(* CODESYS project CodesysJsonParser

Project tree, tasks and I/O mapping:
  Device : ctrlX CORE x64, Bosch Rexroth AG, version 3.6.3.0
    application Application
      libraries: ; ADT, 1.0.0 (Open Source); FloatingPointUtils, 3.5.17.0 (System)
      task MainTask (cyclic, interval 10 ms, priority 30) calls PLC_PRG
      CheckFunctions/
        function CheckBounds [ST]
        function CheckDivDInt [ST]
        function CheckDivLInt [ST]
        function CheckDivLReal [ST]
        function CheckDivReal [ST]
        function CheckLRangeSigned [ST]
        function CheckLRangeUnsigned [ST]
        function CheckPointer [ST]
        function CheckRangeSigned [ST]
        function CheckRangeUnsigned [ST]
      DynamicInterfaces (Not Yet Tested)/
        interface iDynamicDataContainer
        interface iDynamicHashTable
      function GetJsonNodeByKey2 [ST]
      function GetJsonNodeByKey [ST]
      function GetNextJsonToken [ST]
      function GetNodeAsBool [ST]
      function GetNodeAsInt [ST]
      function GetNodeAsObject [ST]
      function GetNodeAsReal [ST]
      function GetNodeAsString [ST]
      function GetNodeAtIndex [ST]
      function GetSubString [ST]
      data type HashData
      function isJsonNodeNull [ST]
      Json/
        function block FB_JsonDomParser [ST]: CopyJson, CopyString, FindMember, GetArrayValueByIdx, GetBool, GetInt, GetString, ParseDocument
        function block FB_JsonSaxWriter [ST]: AddBool, AddDint, AddKey, AddNull, AddString, AddUdint, CopyDocument, EndArray, EndObject, FB_Exit, Init, ResetDocument, StartArray, StartObject
        Types/
      data type JsonDataType
      function block JsonDomParser [ST]: CopyJson, CopyString, FB_Exit, FindMember, GetArrayValueByIdx, GetBool, GetInt, GetReal, GetString, isNull, ParseDocument, ResetDocument
      function JsonHadlr [ST]
      data type JsonObject
      function block JsonParser2 [ST]: CreateJsonType, DeleteJsonNode, FB_Exit, GetRootDoc, Parse, Clean, CreateArray, CreateObj
      function block JsonParser [ST]: Clean, DeleteJsonNode, FB_Exit, GetRootDoc, Parse
      function block JsonSaxWriter [ST]: AddBool, AddChild, AddDint, AddFloat, AddKey, AddNull, AddString, AddUdint, Clean, CopyDocument, CreateArray, CreateJsonType, CreateObj, DeleteJsonNode, EndArray, EndObject, GetRoot, Init, ResetDocument, StartArray, StartObject
      data type JsonSerializeConfig
      data type JsonToken
      data type JsonTokenType
      data type JsonType
      global variables Parameters
      data type pDoc
      program PLC_PRG [ST]
      data type pVoid
      ResizableMem (Not Fully Tested)/
        function block DynamicHashContainer [ST]: CopyToNew, EndResize, FB_Exit, Get, GetNew, GetNewPointer, GetPointer, GetSize, Put, StartResize, FB_Init
        function block DynamicHashTable [ST]: EndResize
        function block DynamicMap [ST]: Remove, Get, HasKey, Put, Resize, Size
        function block DynamicQueue [ST]
        function block DynamicStringContainer [ST]: FB_Exit, CopyToNew, EndResize, Get, GetNew, GetNewPointer, GetPointer, Put
        function block JsonListManager [ST]: Create, Destroy, GetAt, Push
        function block DynamicJsonContainerContainer [ST]: CopyToNew, EndResize, FB_Exit, Get, GetNew, GetNewPointer, GetPointer, GetSize, Put, FB_Init, StartResize
        function block DynamicJsonObjectContainer [ST]: CopyToNew, FB_Exit, Get, GetNew, GetNewPointer, GetPointer, Put, EndResize, FB_Init, GetSize, StartResize
        function block DynamicJsonTypeContainer [ST]: CopyToNew, EndResize, FB_Init, Get, GetNew, GetNewPointer, GetPointer, Put, FB_Exit, GetSize, StartResize
        function block DynamicList [ST]: Get, GetPointer, Insert, Pop, PopBack, PopFront, PushBack, PushFront, Put, Remove, Resize
        global variables JsonHelpers
        function block JsonObjectManager [ST]: Create, Destroy, GetKeyAtIndex, GetValue, Put, Size, FB_Exit
      Serialize/
        function JsonSerializer [ST]
        function SerializeJsonValue [ST]
        function WriteDint [ST]
        function WriteNewLine [ST]
        function WriteReal [ST]
        global variables SerializerConstants
        function WriteByte [ST]
        function WriteColon [ST]
        function WriteEscapedString [ST]
        function WriteIndent [ST]
      Symbols
      Util/
        function block ADT_CompareString [ST]: Compare
        function block StringHash [ST]: Hash
    Realtime_Data : DataLayer, Bosch Rexroth AG, version 3.6.2.0
  commdata.all
  JsonST.Sync
*)

// Device/Application/HashData
{attribute 'enable_dynamic_creation'}
(*Data to keep track of Hash Table to ensure collisions are handled gracefully*)
TYPE HashData :
STRUCT
	isOccupied : BOOL; 
	isDeleted  : BOOL; 
END_STRUCT
END_TYPE

// Device/Application/JsonDataType
TYPE JsonDataType :
(
    JSON_DATA_NULL,
    JSON_DATA_BOOL,
    JSON_DATA_INT,
    JSON_DATA_REAL,
    JSON_DATA_STRING,
    JSON_DATA_ARRAY,
    JSON_DATA_OBJECT
);
END_TYPE

// Device/Application/JsonObject
{attribute 'enable_dynamic_creation'}
TYPE JsonObject :
STRUCT
	pKeys   : POINTER TO POINTER TO JsonType; 
	pValues : POINTER TO  POINTER TO JsonType; 
	iNumValues : INT; 
END_STRUCT
END_TYPE

// Device/Application/JsonSerializeConfig
TYPE JsonSerializeConfig :
STRUCT
    PrettyPrint  : BOOL;        // Enable pretty printing
    IndentLevel  : DINT;        // Current indentation depth (pass 0 initially)
    IndentSize   : DINT;        // Number of spaces per indent level
END_STRUCT
END_TYPE

// Device/Application/JsonToken
TYPE JsonToken :
STRUCT
	TokenType : JsonTokenType;
    StartIndex : LINT;
    Length : DINT;
END_STRUCT
END_TYPE

// Device/Application/JsonTokenType
TYPE JsonTokenType :
(
	JSON_TOKEN_NULL,
    JSON_TOKEN_TRUE,
    JSON_TOKEN_FALSE,
    JSON_TOKEN_NUMBER,
    JSON_TOKEN_STRING,
    JSON_TOKEN_LBRACE,      // {
    JSON_TOKEN_RBRACE,      // }
    JSON_TOKEN_LBRACKET,    // [
    JSON_TOKEN_RBRACKET,    // ]
    JSON_TOKEN_COMMA,       // ,
    JSON_TOKEN_COLON,       // :
    JSON_TOKEN_EOF,
    JSON_TOKEN_ERROR
);
END_TYPE

// Device/Application/JsonType
{attribute 'enable_dynamic_creation'}
TYPE JsonType :
STRUCT
	DataType : JsonDataType; 
	pValue   : pVoid; 
END_STRUCT
END_TYPE

// Device/Application/pDoc
TYPE pDoc : __XWORD; END_TYPE

// Device/Application/pVoid
{attribute 'enable_dynamic_creation'}
TYPE pVoid : __XWORD; END_TYPE

// Device/Application/Parameters
{attribute 'qualified_only'}
VAR_GLOBAL CONSTANT
	MAX_DOC_DEPTH : INT := 50; 
	MAX_ARR_SIZE : INT := 50; 
END_VAR

// Device/Application/ResizableMem (Not Fully Tested)/JsonHelpers
{attribute 'qualified_only'}
VAR_GLOBAL
	instStrCompare     : ADT_CompareString; 
	instStrHash        : StringHash; 
END_VAR

// Device/Application/Serialize/SerializerConstants
{attribute 'qualified_only'}
VAR_GLOBAL CONSTANT
	INDENT_CHAR : BYTE := 32;   // space
    INDENT_SIZE : DINT := 4;    // 4 spaces per level
    NEWLINE_CR  : BYTE := 13;   // \r
    NEWLINE_LF  : BYTE := 10;   // \n
    QUOTE       : BYTE := 34;   // "
    BACKSLASH   : BYTE := 92;   // \
    COLON       : BYTE := 58;   // :
    COMMA       : BYTE := 44;   // ,
    NULL_TERM   : BYTE := 0;    // null terminator
	START_OBJ    : BYTE := 123; 
	END_OBJ      : BYTE := 125; 
	START_ARR    : BYTE := 91; 
	END_ARR      : BYTE := 93;
END_VAR

// Device/Application/PLC_PRG
PROGRAM PLC_PRG
VAR
	Parser : JsonParser2; 
	jsonInput: STRING(8192) := '{"name":"Test","value":42,"active":true, "RealValue" : 12.8, "arrTest" : [[10,11,15][10,11,12]], "subObject" : {"subVal" : 10}}';
	pJson: POINTER TO JsonType;
	pDoc : POINTER TO JsonObject; 
	bVal: BOOL;
	strVal : STRING; 
	size: UDINT;
	iValue: LINT;
	rValue: REAL;
	pJsonAr: POINTER TO JsonType;
	val2: DINT;
	pDoc2 : POINTER TO JsonObject; 
	iVal3: DINT;
	pJsonObject: POINTER TO JsonObjectManager;
	pDint: POINTER TO DINT;
	pByte: Pointer TO Byte;
	pDint2: POINTER TO DINT;
	JsonSettings : JsonSerializeConfig; 
	jSonString : STRING(1000);
	jSonString2 : STRING(1000); 
	Writer : JsonSaxWriter; 
END_VAR

Parser.Parse(ADR(jsonInput),SIZEOF(jsonInput));
pDoc := Parser.GetRootDoc(); 
pJson := GetJsonNodeByKey2('active', pDoc := pDoc); 
GetNodeAsBool(pJson, bJsonVal => bVal); 
pJson := GetJsonNodeByKey2('name',pDoc := pDoc); 
GetNodeAsString(pJson, ADR(strVal),SIZEOF(strVal),retStrSize => size); 
pJson := GetJsonNodeByKey2('value',pDoc); 
GetNodeAsInt(pJson, iJsonVal => iValue); 
pJson := GetJsonNodeByKey2('RealValue',pDoc);
GetNodeAsReal(pJson, rJsonVal => rValue); 
pJson := GetJsonNodeByKey2('arrTest',pDoc); 
pJsonAr := GetNodeAtIndex(pJson,1); 
pJsonAr := GetNodeAtIndex(pJsonAr,2); 
GetNodeAsInt(pJsonAr, iJsonVal => val2); 
pDOC2 := GetJsonNodeByKey2('subObject', pDoc := pDoc);  
pJson := GetJsonNodeByKey2('subVal', pDoc := pDoc2); 
GetNodeAsInt(pJson, iJsonVal => iVal3); 

JsonSettings.IndentSize := 4; 
JsonSettings.PrettyPrint := TRUE; 
JsonSerializer(pDOc, ADR(jSonString),SIZEOF(JsonString),JsonSettings); 
Parser.Clean();
Writer.StartObject(); 
Writer.AddKey('test_bool'); 
Writer.AddBool(TRUE); 
Writer.AddKey('test_dint'); 
Writer.AddDint(100); 
Writer.AddKey('test_real'); 
Writer.AddFloat(90.2); 
Writer.AddKey('test_null'); 
Writer.AddNull(); 
Writer.AddKey('test_string'); 
Writer.AddString('test string val'); 
Writer.AddKey('test_arr'); 
Writer.StartArray(); 
	Writer.StartArray();
		Writer.AddDint(1); 
		Writer.AddDint(2); 
		Writer.AddDint(3);
	Writer.EndArray(); 
	Writer.StartArray(); 
		Writer.AddDint(4); 
		Writer.AddDint(5); 
		Writer.AddDint(6); 
	Writer.EndArray();  
Writer.EndArray(); 
Writer.AddKey('test_obj'); 
Writer.StartObject(); 
	Writer.AddKey('test_internal_object');
	Writer.StartObject(); 
		Writer.AddKey('test_obj_val'); 
		Writer.AddString('obj_val'); 
		Writer.AddKey('test2'); 
		Writer.AddDint(1); 
	Writer.EndObject(); 
	Writer.AddKey('test_internal_object2');
	Writer.StartObject(); 
		Writer.AddKey('test_obj_val'); 
		Writer.AddString('obj_val2'); 
		Writer.AddKey('test2'); 
		Writer.AddDint(2); 
	Writer.EndObject(); 
Writer.EndObject(); 
Writer.CopyDocument(pDoc := JsonString2, nDoc := SIZEOF(JsonString2),bPretty := TRUE); 
Writer.ResetDocument();

END_PROGRAM

// Device/Application/GetJsonNodeByKey2
FUNCTION GetJsonNodeByKey2: Pointer TO JsonType; 
VAR_INPUT
	strKey : STRING; 
END_VAR
VAR_IN_OUT
	pDoc : POINTER TO JsonType; 
END_VAR
VAR_OUTPUT
END_VAR
VAR
	i: INT;
	pStr : POINTER TO STRING; 
	pJsonObject : Pointer TO JsonObjectManager; 
END_VAR

GetJsonNodeByKey2 := 0; 
IF pDoc = 0 THEN 
	RETURN; 
END_IF
IF pDoc^.DataType <> JsonDataType.JSON_DATA_OBJECT THEN 
	RETURN; 
END_IF
pJsonObject := pDoc^.pValue; 
IF pJsonObject <> 0 THEN 
	GetJsonNodeByKey2 := pJsonObject^.GetValue(strKey); 
END_IF

END_FUNCTION

// Device/Application/ResizableMem (Not Fully Tested)/JsonObjectManager
{attribute 'enable_dynamic_creation'}
FUNCTION_BLOCK JsonObjectManager
VAR_INPUT
END_VAR
VAR
	_KeyBacking: POINTER TO DynamicStringContainer;
	_HashBacking: POINTER TO DynamicHashContainer;
	_ValueContainer: POINTER TO DynamicJsonTypeContainer;
	_HashTable: POINTER TO DynamicHashTable;
	_DynamicMap: POINTER TO DynamicMap;
	_KeysListBacking : POINTER TO DynamicStringContainer; 
	_lKeys           : POINTER TO DynamicList;
END_VAR

METHOD Create : BOOL
VAR_INPUT
END_VAR
IF _KeyBacking <> 0 THEN 
	RETURN; 
END_IF
_KeyBacking := __NEW(DynamicStringContainer(udSize := 3)); 
_HashBacking := __NEW(DynamicHashContainer(udSize :=3)); 
_ValueContainer := __NEW(DynamicJsonTypeContainer(udSize :=3)); 
_HashTable := __NEW(DynamicHashTable()); 
_HashTable^(KeyContainer := _KeyBacking^, HashDataContainer := _HashBacking^, Compareator := JsonHelpers.instStrCompare, Hasher := JsonHelpers.instStrHash); 
_DynamicMap := __NEW(DynamicMap); 
_DynamicMap^(KeyContainer := _HashTable^, ValueContainer := _ValueContainer^); 

_KeysListBacking := __NEW(DynamicStringContainer(udSize := 3));  
_lKeys           := __NEW(DynamicList); 
_lKeys^(DataContainer :=_KeysListBacking^);
END_METHOD

METHOD Destroy : BOOL
VAR_INPUT
END_VAR
IF (_KeyBacking <> 0 ) THEN 
	__DELETE(_KeyBacking);
END_IF
IF _HashBacking <> 0 THEN 
__DELETE(_HashBacking); 
END_IF
IF _ValueContainer <> 0 THEN 
__DELETE(_ValueContainer);
END_IF
IF _HashTable <> 0 THEN   
__DELETE(_HashTable); 
END_IF
IF _DynamicMap <> 0 THEN 
__DELETE(_DynamicMap); 
END_IF
IF _lKeys <> 0 THEN 
	__DELETE(_lKeys); 
END_IF
IF _KeysListBacking <> 0 THEN
	__DELETE(_KeysListBacking);
END_IF
END_METHOD

METHOD GetKeyAtIndex : Pointer TO STRING
VAR_INPUT
	index : UDINT; 
END_VAR
VAR
	pString : POINTER TO STRING; 
END_VAR
_lKeys^.Get(index,ADR(pString)); 
GetKeyAtIndex := pString;
END_METHOD

METHOD GetValue : POINTER TO JsonType
VAR_INPUT
	stKey  : STRING; 
END_VAR
VAR
	pJsonValue : POINTER TO JsonType;  
	pString : POINTER TO STRING; 
	ppString : POINTER TO POINTER TO STRING; 
END_VAR
GetValue := 0; 
pString := ADR(stKey); 
ppSTring := ADR(pString); 
IF _DynamicMap <> 0 THEN
	_DynamicMap^.Get(ppstring, ADR(pJsonValue)); 
	GetValue := pJsonValue; 
END_IF
END_METHOD

METHOD Put : BOOL
VAR_INPUT
	pString : POINTER TO BYTE; 
	pValue  : Pointer TO JsonType; 
END_VAR
Put := FALSE; 
IF _DynamicMap = 0 THEN 
	RETURN;
END_IF
IF(_DynamicMap^.Put(pKey := ADR(pString), pValue := ADR(pValue))) THEN
	_lKeys^.PushBack(ADR(pString));
	Put := TRUE;  
END_IF
END_METHOD

PROPERTY Size : UDINT
GET
IF _lKeys <> 0 THEN
	Size := _lKeys^.Size;
ELSE
	Size := 0; 
END_IF;
END_GET
END_PROPERTY

//FB_Exit must be implemented explicitly. If there is an implementation, then the
//method is called before the controller removes the code of the function block instance
//(implicit call). The return value is not evaluated.
METHOD FB_Exit: BOOL
VAR_INPUT
    bInCopyCode: BOOL;  // TRUE: the exit method is called in order to leave the instance which will be copied afterwards (online change).  
END_VAR
Destroy();
END_METHOD

END_FUNCTION_BLOCK

// Device/Application/ResizableMem (Not Fully Tested)/DynamicStringContainer
{attribute 'enable_dynamic_creation'}
FUNCTION_BLOCK DynamicStringContainer IMPLEMENTS iDynamicDataContainer
VAR_INPUT
	udSize : UDINT; 
END_VAR
VAR_OUTPUT
END_VAR
VAR
	_ptrBackingArray : POINTER TO POINTER TO BYTE;
	_ptrTempNewArray : POINTER TO POINTER TO BYTE;  
	_size : UDINT; 
	_tData : POINTER TO BYTE; 
	_pData : POINTER TO POINTER TO BYTE; 
	_newSize: UDINT;
	_byteSize : UDINT; 
END_VAR

_byteSize := SIZEOF(_tData); 
_newSize := udSize * _byteSize;
_ptrBackingArray := __NEW(BYTE,_newSize); 
_size := udSize;

//FB_Exit must be implemented explicitly. If there is an implementation, then the
//method is called before the controller removes the code of the function block instance
//(implicit call). The return value is not evaluated.
METHOD FB_Exit: BOOL
VAR_INPUT
    bInCopyCode: BOOL;  // TRUE: the exit method is called in order to leave the instance which will be copied afterwards (online change).  
END_VAR
VAR
	i: UDINT;
END_VAR
IF _ptrBackingArray <> 0 THEN 
	__DELETE(_ptrBackingArray); 
END_IF
IF _ptrTempNewArray <> 0 THEN 
	__DELETE(_ptrTempNewArray); 
END_IF
END_METHOD

{attribute 'no_check'}
METHOD CopyToNew : BOOL
VAR_INPUT
	indexOld	: UDINT;
	indexNew	: UDINT;
END_VAR
CopyToNew := FALSE; 
IF indexOld < _size/2 AND indexNew < _size THEN 
	_ptrTempNewArray[indexNew] := _ptrBackingArray[indexOld]; 
	CopyToNew := TRUE; 
END_IF
END_METHOD

{attribute 'no_check'}
METHOD EndResize : BOOL
__DELETE(_ptrBackingArray); 
_ptrBackingArray := _ptrTempNewArray; 
_ptrTempNewArray := 0;
END_METHOD

{attribute 'no_check'}
METHOD Get : BOOL
VAR_INPUT
	index	: UDINT;
	pData	: PVoid;
END_VAR
IF index < _size THEN 
	_pData := pData; 
	_pData^ := _ptrBackingArray[index]; 
	GET := TRUE; 
ELSE 
	GET := FALSE; 
END_IF
END_METHOD

{attribute 'no_check'}
METHOD GetNew : BOOL
VAR_INPUT
	index	: UDINT;
	pData	: PVoid;
END_VAR
IF _ptrTempNewArray <> 0 AND index < _size THEN 
	_pData := pData; 
	_pData^ :=_ptrTempNewArray[index]; 
	GetNew := TRUE; 
ELSE 
	GetNew := FALSE; 
END_IF
END_METHOD

{attribute 'no_check'}
METHOD GetNewPointer : PVoid
VAR_INPUT
	index	: UDINT;
END_VAR
IF _ptrTempNewArray <> 0 AND index < _size THEN 
	GetNewPointer := ADR(_ptrTempNewArray[index]); 
ELSE 
	GetNewPointer := 0; 
END_IF
END_METHOD

{attribute 'no_check'}
METHOD GetPointer : PVoid
VAR_INPUT
	index	: UDINT;
END_VAR
IF index < _size THEN 
	GetPointer := ADR(_ptrBackingArray[index]); 
ELSE 
	GetPointer := 0; 
END_IF
END_METHOD

{attribute 'no_check'}
METHOD Put : BOOL
VAR_INPUT
	index	: UDINT;
	pData	: PVoid;
END_VAR
_pData := pData; 
Put := FALSE; 
IF index < _size THEN 
	_ptrBackingArray[index] := _pData^; 
	Put := TRUE; 
END_IF
END_METHOD

END_FUNCTION_BLOCK

// Device/Application/DynamicInterfaces (Not Yet Tested)/iDynamicDataContainer
INTERFACE iDynamicDataContainer Extends iDataContainer;

END_INTERFACE

// Device/Application/ResizableMem (Not Fully Tested)/DynamicHashContainer
{attribute 'enable_dynamic_creation'}
FUNCTION_BLOCK DynamicHashContainer IMPLEMENTS iDynamicDataContainer
VAR_INPUT
	udSize : UDINT; 
END_VAR
VAR_OUTPUT
END_VAR
VAR
	_ptrBackingArray : POINTER TO BYTE;
	_ptrTempNewArray : POINTER TO BYTE;  
	_size : UDINT; 
	_tData : ADT.HashData; 
	_pData : POINTER TO ADT.HashData; 
	_newSize: UDINT;
	_byteSize : UDINT; 
	_i: UDINT;
END_VAR

_byteSize := 1; 
 _newSize := udSize;
_ptrBackingArray := __NEW(BYTE,_newSize);
FOR _i := 0 TO _newSize DO
	_ptrBackingArray[_i] := 0; 
END_FOR 
_size := udSize;

METHOD CopyToNew : BOOL
VAR_INPUT
	indexOld	: UDINT;
	indexNew	: UDINT;
END_VAR
CopyToNew := FALSE; 
IF indexOld < _size/2 AND indexNew < _size THEN 
	_ptrTempNewArray[indexNew] := _ptrBackingArray[indexOld]; 
	CopyToNew := TRUE; 
END_IF
END_METHOD

METHOD EndResize : BOOL
__DELETE(_ptrBackingArray); 
_ptrBackingArray := _ptrTempNewArray; 
_ptrTempNewArray := 0;
END_METHOD

//FB_Exit must be implemented explicitly. If there is an implementation, then the
//method is called before the controller removes the code of the function block instance
//(implicit call). The return value is not evaluated.
METHOD FB_Exit: BOOL
VAR_INPUT
    bInCopyCode: BOOL;  // TRUE: the exit method is called in order to leave the instance which will be copied afterwards (online change).  
END_VAR
VAR
	i: UDINT;
END_VAR
IF _ptrBackingArray <> 0 THEN 
	__DELETE(_ptrBackingArray); 
END_IF
IF _ptrTempNewArray <> 0 THEN 
	__DELETE(_ptrTempNewArray); 
END_IF
END_METHOD

METHOD Get : BOOL
VAR_INPUT
	index	: UDINT;
	pData	: PVoid;
END_VAR
IF index < _size THEN 
	_pData := pData; 
	_pData^.isOccupied := _ptrBackingArray[index].0; 
	_pData^.isDeleted :=  _ptrBackingArray[index].1; 
	GET := TRUE; 
ELSE 
	GET := FALSE; 
END_IF
END_METHOD

METHOD GetNew : BOOL
VAR_INPUT
	index	: UDINT;
	pData	: PVoid;
END_VAR
IF _ptrTempNewArray <> 0 AND index < _size THEN 
	_pData := pData; 
	_pData^.isOccupied :=_ptrTempNewArray[index].0; 
	_pData^.isDeleted  := _ptrTempNewArray[index].1; 
	GetNew := TRUE; 
ELSE 
	GetNew := FALSE; 
END_IF
END_METHOD

METHOD GetNewPointer : PVoid
VAR_INPUT
	index	: UDINT;
END_VAR
IF _ptrTempNewArray <> 0 AND index < _size THEN 
	GetNewPointer := ADR(_ptrTempNewArray[index]); 
ELSE 
	GetNewPointer := 0; 
END_IF
END_METHOD

METHOD GetPointer : PVoid
VAR_INPUT
	index	: UDINT;
END_VAR
IF index < _size THEN 
	GetPointer := ADR(_ptrBackingArray[index]); 
ELSE 
	GetPointer := 0; 
END_IF
END_METHOD

METHOD GetSize : UDINT
GetSize :=_size;
END_METHOD

METHOD Put : BOOL
VAR_INPUT
	index	: UDINT;
	pData	: PVoid;
END_VAR
_pData := pData; 
Put := FALSE; 
IF index < _size THEN 
	_ptrBackingArray[index].0 := _pData^.isOccupied; 
	_ptrBackingArray[index].1 := _pData^.isDeleted; 
	Put := TRUE; 
END_IF
END_METHOD

METHOD StartResize : BOOL
VAR
	_newSize: UDINT;
	_i: LINT;
END_VAR
_newSize := (2* _size)*_byteSize;
_ptrTempNewArray := __NEW(BYTE,_newSize); 
_size := _size * 2; 
FOR _i := 0 TO _size - 1 DO 
	_ptrTempNewArray[_i] := 0; 
END_FOR
END_METHOD

//FB_Init is always available implicitly and it is used primarily for initialization.
//The return value is not evaluated. For a specific influence, you can also declare the
//methods explicitly and provide additional code there with the standard initialization
//code. You can evaluate the return value.
METHOD FB_Init: BOOL
VAR_INPUT
    bInitRetains: BOOL; // TRUE: the retain variables are initialized (reset warm / reset cold)
    bInCopyCode: BOOL;  // TRUE: the instance will be copied to the copy code afterward (online change) 
	udSize      : UDINT;   
END_VAR
this^(udSize := udSize);
END_METHOD

END_FUNCTION_BLOCK

// Device/Application/ResizableMem (Not Fully Tested)/DynamicJsonTypeContainer
{attribute 'enable_dynamic_creation'}
FUNCTION_BLOCK DynamicJsonTypeContainer IMPLEMENTS iDynamicDataContainer
VAR_INPUT
	udSize : UDINT; 
END_VAR
VAR_OUTPUT
END_VAR
VAR
	_ptrBackingArray : POINTER TO POINTER TO JsonType;
	_ptrTempNewArray : POINTER TO POINTER TO JsonType;  
	_size : UDINT; 
	_tData : POINTER TO JsonType; 
	_pData : POINTER TO POINTER TO JsonType; 
	_newSize: UDINT;
	_byteSize : UDINT; 
END_VAR

_byteSize := SIZEOF(_tData); 
_newSize := udSize * _byteSize;
_ptrBackingArray := __NEW(BYTE,_newSize); 
_size := udSize;

METHOD CopyToNew : BOOL
VAR_INPUT
	indexOld	: UDINT;
	indexNew	: UDINT;
END_VAR
CopyToNew := FALSE; 
IF indexOld < _size/2 AND indexNew < _size THEN 
	_ptrTempNewArray[indexNew] := _ptrBackingArray[indexOld]; 
	CopyToNew := TRUE; 
END_IF
END_METHOD

METHOD EndResize : BOOL
__DELETE(_ptrBackingArray); 
_ptrBackingArray := _ptrTempNewArray; 
_ptrTempNewArray := 0;
END_METHOD

//FB_Init is always available implicitly and it is used primarily for initialization.
//The return value is not evaluated. For a specific influence, you can also declare the
//methods explicitly and provide additional code there with the standard initialization
//code. You can evaluate the return value.
METHOD FB_Init: BOOL
VAR_INPUT
    bInitRetains: BOOL; // TRUE: the retain variables are initialized (reset warm / reset cold)
    bInCopyCode: BOOL;  // TRUE: the instance will be copied to the copy code afterward (online change) 
	udSize      : UDINT;   
END_VAR
this^(udSize := udSize);
END_METHOD

METHOD Get : BOOL
VAR_INPUT
	index	: UDINT;
	pData	: PVoid;
END_VAR
IF index < _size THEN 
	_pData := pData; 
	_pData^ := _ptrBackingArray[index]; 
	GET := TRUE; 
ELSE 
	GET := FALSE; 
END_IF
END_METHOD

METHOD GetNew : BOOL
VAR_INPUT
	index	: UDINT;
	pData	: PVoid;
END_VAR
IF _ptrTempNewArray <> 0 AND index < _size THEN 
	_pData := pData; 
	_pData^ :=_ptrTempNewArray[index]; 
	GetNew := TRUE; 
ELSE 
	GetNew := FALSE; 
END_IF
END_METHOD

METHOD GetNewPointer : PVoid
VAR_INPUT
	index	: UDINT;
END_VAR
IF _ptrTempNewArray <> 0 AND index < _size THEN 
	GetNewPointer := ADR(_ptrTempNewArray[index]); 
ELSE 
	GetNewPointer := 0; 
END_IF
END_METHOD

METHOD GetPointer : PVoid
VAR_INPUT
	index	: UDINT;
END_VAR
IF index < _size THEN 
	GetPointer := ADR(_ptrBackingArray[index]); 
ELSE 
	GetPointer := 0; 
END_IF
END_METHOD

METHOD Put : BOOL
VAR_INPUT
	index	: UDINT;
	pData	: PVoid;
END_VAR
_pData := pData; 
Put := FALSE; 
IF index < _size THEN 
	_ptrBackingArray[index] := _pData^; 
	Put := TRUE; 
END_IF
END_METHOD

//FB_Exit must be implemented explicitly. If there is an implementation, then the
//method is called before the controller removes the code of the function block instance
//(implicit call). The return value is not evaluated.
METHOD FB_Exit: BOOL
VAR_INPUT
    bInCopyCode: BOOL;  // TRUE: the exit method is called in order to leave the instance which will be copied afterwards (online change).  
END_VAR
VAR
	i: UDINT;
END_VAR
IF _ptrBackingArray <> 0 THEN 
	__DELETE(_ptrBackingArray); 
END_IF
IF _ptrTempNewArray <> 0 THEN 
	__DELETE(_ptrTempNewArray); 
END_IF
END_METHOD

METHOD GetSize : UDINT
GetSize :=_size;
END_METHOD

METHOD StartResize : BOOL
VAR
	_newSize: UDINT;
END_VAR
_newSize := (2* _size)*_byteSize;
_ptrTempNewArray := __NEW(BYTE,_newSize); 
_size := _size * 2;
END_METHOD

END_FUNCTION_BLOCK

// Device/Application/ResizableMem (Not Fully Tested)/DynamicHashTable
{attribute 'no_check'}
{attribute 'enable_dynamic_creation'}
FUNCTION_BLOCK DynamicHashTable IMPLEMENTS iDynamicHashTable
VAR_INPUT
	KeyContainer : iDynamicDataContainer;
	HashDataContainer : iDynamicDataContainer;  
	Compareator : iCompare;
	Hasher      : iHash;  
END_VAR
VAR_OUTPUT
END_VAR
VAR
END_VAR

METHOD EndResize : BOOL
KeyContainer.EndResize(); 
HashDataContainer.EndResize();
END_METHOD

END_FUNCTION_BLOCK

// Device/Application/DynamicInterfaces (Not Yet Tested)/iDynamicHashTable
INTERFACE iDynamicHashTable EXTENDS iDynamicDataContainer,iCompare,iHash

END_INTERFACE

// Device/Application/ResizableMem (Not Fully Tested)/DynamicMap
{attribute 'no_check'}
{attribute 'enable_dynamic_creation'}
FUNCTION_BLOCK DynamicMap IMPLEMENTS iMap
VAR_INPUT
	KeyContainer : iDynamicHashTable; 
	ValueContainer : iDynamicDataContainer;  
END_VAR
VAR_OUTPUT
END_VAR
VAR
	_backingSize : UDINT := 0;
	_size : DINT := 0;  
END_VAR

{attribute 'no_check'}
METHOD Remove : BOOL
VAR_INPUT
	pKey	: pVoid;
END_VAR

VAR
	hash: LINT;
	index: UDINT;
	_i: UDINT;
	_tIndex: UDINT;
	pData: ADT.PVoid;
	pOldKey: ADT.PVoid;
END_VAR
Remove := FALSE; 
IF(_backingSize = 0 ) THEN 
	_backingSize := KeyContainer.GetSize(); 
END_IF
hash :=  KeyContainer.Hash(pKey); 
index := LINT_TO_UDINT(hash MOD _backingSize); 
WHILE _i < _backingSize - 1 DO 
	_tIndex := (_i + index) MOD _backingSize; 
	IF NOT (KeyContainer.isOccupied(_tIndex) OR KeyContainer.isDeleted(_tIndex))THEN 
		EXIT; 
	END_IF
	IF KeyContainer.Compare(pKey, KeyContainer.GetNewPointer(_tIndex)) = 0 THEN 
		KeyContainer.Delete(_tIndex);  
		Remove := TRUE; 
		_size := _size -1; 
		EXIT; 
	END_IF
	_i := _i+ 1; 
END_WHILE
END_METHOD

{attribute 'no_check'}
METHOD Get : BOOL
VAR_INPUT
	pKey	: pVoid;
	pValue	: pVoid;
END_VAR

VAR
	hash: LINT;
	index: UDINT;
	_i : UDINT; 
	_tIndex: UDINT;
END_VAR
Get := FALSE; 
IF(_backingSize = 0 ) THEN 
	_backingSize := KeyContainer.GetSize(); 
END_IF
hash :=  KeyContainer.Hash(pKey); 
index := LINT_TO_UDINT(hash MOD _backingSize); 
WHILE _i < _backingSize  DO 
	_tIndex := (_i + index) MOD _backingSize; 
	IF NOT (KeyContainer.isOccupied(_tIndex) OR KeyContainer.isDeleted(_tIndex))THEN 
		EXIT; 
	END_IF
	IF KeyContainer.Compare(pKey, KeyContainer.GetPointer(_tIndex)) = 0 THEN 
		ValueContainer.Get(_tIndex,pValue); 
		Get := TRUE; 
		EXIT; 
	END_IF
	_i := _i+ 1; 
END_WHILE
END_METHOD

{attribute 'no_check'}
METHOD HasKey : BOOL
VAR_INPUT
	pKey : pVoid; 
END_VAR

VAR
	hash: LINT;
	index: UDINT;
	_i: UDINT;
	_tIndex: UDINT;
END_VAR
HasKey := FALSE; 
IF(_backingSize = 0 ) THEN 
	_backingSize := KeyContainer.GetSize(); 
END_IF
hash :=  KeyContainer.Hash(pKey); 
index := LINT_TO_UDINT(hash MOD _backingSize); 
WHILE _i < _backingSize - 1 DO 
	_tIndex := (_i + index) MOD _backingSize; 
	IF NOT (KeyContainer.isOccupied(_tIndex) OR KeyContainer.isDeleted(_tIndex))THEN 
		EXIT; 
	END_IF
	IF KeyContainer.Compare(pKey, KeyContainer.GetPointer(_tIndex)) = 0 THEN  
		HasKey := TRUE; 
		EXIT; 
	END_IF
	_i := _i+ 1; 
END_WHILE
END_METHOD

{attribute 'no_check'}
METHOD Put : BOOL
VAR_INPUT
	pKey	: pVoid;
	pValue	: pVoid;
END_VAR

VAR
	hash: LINT;
	index: UDINT;
	_i: UDINT;
	_tIndex: UDINT;
END_VAR
Put := FALSE; 
IF(_backingSize = 0 ) THEN 
	_backingSize := KeyContainer.GetSize(); 
END_IF
IF _size >= TO_DINT(0.7 * TO_REAL(_backingSize)) THEN 
	_backingSize := resize(); 
END_IF
hash :=  KeyContainer.Hash(pKey); 
index := LINT_TO_UDINT(hash MOD _backingSize); 
_i:= 0; 
WHILE _i < _backingSize DO 
	_tIndex := (_i + index) MOD _backingSize; 
	IF (KeyContainer.isOccupied(_tIndex)) THEN 
		IF KeyContainer.Compare(pKey, KeyContainer.GetPointer(_tIndex)) = 0 THEN 
			ValueContainer.Put(_tIndex,pValue); 
			PUT := TRUE; 
			EXIT;
		END_IF
	ELSE 
		ValueContainer.Put(_tIndex,pValue); 
		KeyContainer.Put(_tIndex,pKey); 
		PUT := TRUE; 
		_size := _size + 1; 
		EXIT;
	END_IF 	
	_i := _i + 1; 
END_WHILE
END_METHOD

METHOD PRIVATE Resize : UDINT
VAR_INPUT
END_VAR

VAR
	_i: UDINT;
	_newSize: UDINT;
	index: UDINT;
	hash: LINT;
	_tIndex: UDINT;
	_j: UINT;
	pData : pVOID; 
	pKey: PVoid;
END_VAR
ValueContainer.StartResize();
KeyContainer.StartResize(); 
_newSize := KeyContainer.GetSize(); 
FOR _i := 0 TO _backingSize - 1 DO 
	IF KeyContainer.isOccupied(_i) THEN 
		hash :=  KeyContainer.Hash(KeyContainer.GetPointer(_i)); 
		index := LINT_TO_UDINT(hash MOD _newSize); 
		_j := 0; 
		WHILE _j < _backingSize  DO 
			_tIndex := (_j + index) MOD _newSize; 
			IF (KeyContainer.isNewOccupied(_tIndex)) THEN 
				IF KeyContainer.Compare(KeyContainer.GetPointer(_i), KeyContainer.GetNewPointer(_tIndex)) = 0 THEN 
					KeyContainer.CopyToNew(_i,_tindex); 
					ValueContainer.CopyToNew(_i,_tindex); 
					EXIT;
				END_IF
			ELSE 
				KeyContainer.CopyToNew(_i,_tindex); 
				ValueContainer.CopyToNew(_i,_tindex); 
				EXIT;
			END_IF 	
			_j := _j + 1; 
		END_WHILE
	END_IF
END_FOR
Resize := 2*_backingSize; 
ValueContainer.EndResize();
KeyContainer.EndResize();
END_METHOD

PROPERTY Size : DINT
GET
Size := _size;
END_GET
END_PROPERTY

END_FUNCTION_BLOCK

// Device/Application/ResizableMem (Not Fully Tested)/DynamicList
{attribute 'no_check'}
{attribute 'enable_dynamic_creation'}
FUNCTION_BLOCK DynamicList IMPLEMENTS iList
VAR_INPUT
	DataContainer :  iDynamicDataContainer; 
END_VAR
VAR_OUTPUT
END_VAR
VAR
	_size : UDINT; 
	_iterator : Iterator; 
	_bIteratorOpened : BOOL; 
	_backingSize: UDINT;
	_front: UDINT;
END_VAR

{attribute 'no_check'}
METHOD Get : BOOL
VAR_INPUT
	Index	: UDINT;
	pData	: PVOID;
END_VAR
IF _backingSize = 0 THEN 
	_backingSize := DataContainer.GetSize(); 
END_IF
IF Index < _size THEN 
	Get := DataContainer.Get((Index + _front) MOD _backingSize ,pData); 
ELSE 
	Get := FALSE; 
END_IF
END_METHOD

{attribute 'no_check'}
METHOD GetPointer : Bool
VAR_INPUT
	Index	: UDINT;
END_VAR
VAR_OUTPUT
	pData : PVoid; 
END_VAR
IF _backingSize = 0 THEN 
	_backingSize := DataContainer.GetSize(); 
END_IF
IF Index < _size THEN 
	pData := DataContainer.GetPointer((Index + _front) MOD _backingSize);
	GetPointer := TRUE; 
ELSE 
	GetPointer := FALSE; 
END_IF
END_METHOD

{attribute 'no_check'}
METHOD Insert : BOOL
VAR_INPUT
	StartIndex	: UDINT; //Start Index
	Values	: iIterable; //Iterable list of values to insert
END_VAR

VAR
	_i: UDINT;
	_index: UDINT;
	_destIndex: UDINT;
END_VAR
IF _backingSize = 0 THEN 
	_backingSize := DataContainer.GetSize(); 
END_IF
WHILE Values.GetIterator().Size >= (_backingSize - size) DO 
	_backingSize := THIS^.Resize();
END_WHILE
IF StartIndex <= _size AND NOT Values.GetIterator().isBusy THEN 
	IF StartIndex <> _size THEN 
		FOR _i := _size - 1  TO StartIndex BY - 1 DO
			_index := (_front + _i) MOD _backingSize; 
			_destIndex := (_index + Values.GetIterator().Size) MOD _backingSize; 
			DataContainer.Put(_destIndex,DataContainer.GetNewPointer(_index)); 
			IF _i = 0 THEN 
				EXIT; 
			END_IF
		END_FOR
	END_IF
	WHILE Values.GetIterator().Next(DataContainer.GetPointer((StartIndex + _front + _i) MOD _backingSize)) DO 
		_i := _i+1; 
		_size := _size + 1; 
	END_WHILE
	Insert := TRUE; 
ELSE 
	Insert := FALSE; 
END_IF
END_METHOD

{attribute 'no_check'}
METHOD Pop : BOOL
VAR_INPUT
	Index	: UDINT;
	pData	: PVOID;
END_VAR

VAR
	_i: UDINT;
	_index: UDINT;
	_indexPlus1: UDINT;
END_VAR
IF _backingSize = 0 THEN 
	_backingSize := DataContainer.GetSize(); 
END_IF
IF Index < _size THEN 
	Pop := DataContainer.Get((Index + _front) MOD _backingSize,pData); 
	FOR _i := Index TO size -1 DO 
		_index := (_front + _i) MOD _backingSize; 
		_indexPlus1 := (_index + 1) MOD _backingSize; 
		DataContainer.Put(_index,DataContainer.GetPointer(_indexPlus1)); 
		IF _i = 0 THEN 
			EXIT; 
		END_IF
	END_FOR
	_size := _size - 1; 
ELSE 
	Pop := FALSE; 
END_IF
END_METHOD

{attribute 'no_check'}
METHOD PopBack : BOOL
VAR_INPUT
	pData	: PVoid;
END_VAR

VAR
END_VAR
IF _backingSize = 0 THEN 
	_backingSize := DataContainer.GetSize(); 
END_IF
IF _size > 0 THEN 
	PopBack := DataContainer.Get((_front + _size) MOD _backingSize ,pData); 
	_size := _size - 1; 
ELSE 
	PopBack := FALSE; 
END_IF
END_METHOD

{attribute 'no_check'}
METHOD PopFront : BOOL
VAR_INPUT
	pData	: PVoid;
END_VAR
IF _backingSize = 0 THEN 
	_backingSize := DataContainer.GetSize(); 
END_IF
IF _size > 0 THEN 
	PopFront := DataContainer.Get(_front,pData); 
	_size := _size - 1; 
	_front := (_front + 1) MOD _backingSize; 
ELSE 
	PopFront := FALSE; 
END_IF
END_METHOD

{attribute 'no_check'}
METHOD PushBack : BOOL
VAR_INPUT
	pData	: PVOID;
END_VAR
IF _backingSize = 0 THEN 
	_backingSize := DataContainer.GetSize(); 
END_IF
IF _size >= _backingSize THEN 
	_backingSize := THIS^.Resize(); 
END_IF
IF _size < _backingSize THEN 
	PushBack := DataContainer.Put((_front+_size) MOD _backingSize,pData); 
	_size := _size + 1;
ELSE 
	PushBack := FALSE; 
END_IF
END_METHOD

{attribute 'no_check'}
METHOD PushFront : BOOL
VAR_INPUT
	pData	: PVOID;
END_VAR
IF _backingSize = 0 THEN 
	_backingSize := DataContainer.GetSize(); 
END_IF
IF _size >= _backingSize THEN 
	_backingSize := THIS^.Resize(); 
END_IF
IF _size < _backingSize THEN 
	_front := _front -1; 
	IF _front >= _backingSize THEN 
		_front := _backingSize - 1; 
	END_IF
	PushFront := DataContainer.Put(_front,pData); 
	_size := _size + 1; 
ELSE 
	PushFront := FALSE; 
END_IF
END_METHOD

{attribute 'no_check'}
METHOD Put : BOOL
VAR_INPUT
	Index	: UDINT;
	pData	: PVoid;
END_VAR

VAR
	_i: UDINT;
	_index : UDINT;
	_indexSub1 : UDINT; 
END_VAR
IF _backingSize = 0 THEN 
	_backingSize := DataContainer.GetSize(); 
END_IF
IF _size >= _backingSize THEN 
	_backingSize := THIS^.Resize(); 
END_IF
IF _size < _backingSize AND Index <= _size THEN 
	IF Index <> _size THEN 
		FOR _i := _size  TO Index + 1 BY - 1 DO
			_index := (_front + _i) MOD _backingSize; 
			_indexSub1 := _index - 1; 
			IF (_indexSub1 >= _backingSize) THEN 
				_indexSub1 := _backingSize -1; 
			END_IF
			DataContainer.Put(_index,DataContainer.GetPointer(_indexSub1)); 
		END_FOR
	END_IF
	Put := DataContainer.Put((Index + _front)MOD _backingSize,pData); 
	_size := _size + 1; 
ELSE 
	Put := FALSE; 
END_IF
END_METHOD

{attribute 'no_check'}
METHOD Remove : BOOL
VAR_INPUT
	Where	: iCompare;
	pData   : PVoid; 
END_VAR

VAR
	_i: UDINT;
	_j: UDINT;
	_index : UDINT; 
	_indexPlus1 : UDINT; 
END_VAR
Remove := FALSE; 
IF _size = 0 THEN 
	RETURN; 
END_IF
FOR _i := 0 TO _size -1 DO 
	IF Where.Compare(pData,DataContainer.GetPointer((_i + _front) MOD _backingSize)) = 0 THEN 
		FOR _j := _i  TO _size-1 DO 
			_index := (_front + _j) MOD _backingSize; 
			_indexPlus1 := (_index + 1) MOD _backingSize; 
			DataContainer.Put(_index,DataContainer.GetPointer(_indexPlus1)); 
		END_FOR
		_size := _size - 1; 
		Remove := TRUE; 
		EXIT; 
	END_IF;
END_FOR
END_METHOD

{attribute 'no_check'}
METHOD PRIVATE Resize : UDINT
VAR_INPUT
END_VAR

VAR
	_i: UDINT;
END_VAR
DataContainer.StartResize(); 
FOR _i := 0 TO THIS^.Size -1 DO 
	DataContainer.CopyToNew((_front + _i) MOD _backingSize, _i); 
END_FOR
_front := 0; 
DataContainer.EndResize();
Resize := DataContainer.GetSize();
END_METHOD

END_FUNCTION_BLOCK

// Device/Application/GetNodeAsBool
FUNCTION GetNodeAsBool : Bool
VAR_INPUT
	pJsonNode : POINTER TO JSONTYPE; 
END_VAR
VAR_OUTPUT
	bJsonVal : BOOL; 
END_VAR
VAR
	pBool : Pointer TO BOOL; 
END_VAR

GetNodeAsBool := FALSE;
IF pJsonNode = 0 THEN 
	RETURN; 
END_IF
IF pJsonNode^.DataType <> JsonDataType.JSON_DATA_BOOL THEN  
	RETURN; 
END_IF
GetNodeAsBool := TRUE; 
pBool := pJsonNode^.pValue; 
bJsonVal := pBool^;

END_FUNCTION

// Device/Application/GetNodeAsString
FUNCTION GetNodeAsString : BOOL
VAR_INPUT
	pJsonNode : POINTER TO JsonType; 
	pOutString : POINTER TO BYTE; 
	StrSize  :  UDINT; 
END_VAR
VAR_OUTPUT
	retStrSize : UDINT; 
END_VAR
VAR
	pStr : POINTER TO BYTE; 
	i : UDINT; 
END_VAR

GetNodeAsString := FALSE; 
IF pJsonNode = 0 THEN 
	RETURN;
END_IF
IF pJsonNode^.DataType <> JsonDataType.JSON_DATA_STRING THEN 
	RETURN; 
END_IF
GetNodeAsString := TRUE; 
pStr := pJsonNode^.pValue;
i := 0;  
WHILE pStr[i] <> 0 AND i <StrSize - 1 DO 
	pOutString[i] := pStr[i]; 
	i := i + 1; 
END_WHILE
pOutString[i] := 0; 
retStrSize := i ;

END_FUNCTION

// Device/Application/GetNodeAsInt
FUNCTION GetNodeAsInt : BOOL
VAR_INPUT
	pJsonNode: POINTER TO JsonType;
END_VAR
VAR_OUTPUT
	iJsonVal : DINT; 
END_VAR
VAR
	pInt : POINTER TO DINT; 
END_VAR

GetNodeAsInt := FALSE; 
IF pJsonNode = 0 THEN 
	RETURN; 
END_IF

IF pJsonNode^.DataType <> JsonDataType.JSON_DATA_INT THEN 
	RETURN; 
END_IF
GetNodeAsInt := TRUE; 
pInt := pJsonNode^.pValue; 
iJsonVal := pInt^;

END_FUNCTION

// Device/Application/GetNodeAsReal
FUNCTION GetNodeAsReal : BOOL
VAR_INPUT
	pJsonNode : POINTER TO JsonType; 
END_VAR
VAR_OUTPUT
	rJsonVal : REAL; 
END_VAR
VAR
	pVal : POINTER TO REAL; 
END_VAR

GetNodeAsReal := FALSE; 
IF pJsonNode = 0 THEN 
	RETURN; 
END_IF

IF pJsonNode^.DataType <> JsonDataType.JSON_DATA_REAL THEN 
	RETURN; 
END_IF
GetNodeAsReal := TRUE; 
pVal := pJsonNode^.pValue; 
rJsonVal := pVal^;

END_FUNCTION

// Device/Application/GetNodeAtIndex
FUNCTION GetNodeAtIndex : POINTER TO JsonType
VAR_INPUT
	pJsonType : POINTER TO JsonType;
	i : UDINT; 
END_VAR

VAR
	pJsonArray : POINTER TO DynamicList; 
	pJsonValue : POINTER TO JsonType;
END_VAR

GetNodeAtIndex := 0; 
IF pJsonType = 0 THEN 
	RETURN; 
END_IF
IF pJsonType^.DataType <> JsonDataType.JSON_DATA_ARRAY THEN 
	RETURN; 
END_IF
pJsonArray := pJsonType^.pValue; 
pJsonArray^.Get(i,ADR(pJsonValue)); 
GetNodeAtIndex := pJsonValue;

END_FUNCTION

// Device/Application/Serialize/JsonSerializer
FUNCTION JsonSerializer : DINT
VAR_INPUT
	root : POINTER TO JSONType; 
	pDest : POINTER TO BYTE; 
	DestSize : DINT; 
END_VAR
VAR_IN_OUT
	Settings : JsonSerializeConfig; 
END_VAR
VAR_OUTPUT
END_VAR
VAR
	arrObjects : ARRAY[0..Parameters.MAX_DOC_DEPTH] OF POINTER TO JsonObjectManager; 
	arrArrays  : ARRAY[0..Parameters.MAX_DOC_DEPTH] OF POINTER TO DynamicList; 
	objIdx : INT; 
	arrIdx : INT; 
	curArrIdx : ARRAY[0.. Parameters.MAX_DOC_DEPTH] OF UDINT;
	curObjIdx : ARRAY[0.. Parameters.MAX_DOC_DEPTH] OF UDINT; 
	pCurJsonVal : POINTER TO JsonType; 
	Offset : DINT; 
	pKey   : POINTER TO STRING;   
	_i: DINT;
	_indentNo: DINT;
END_VAR

JsonSerializer := 0; 
IF root = 0 THEN 
	RETURN; 
END_IF
IF root^.pValue = 0 THEN 
	RETURN; 
END_IF
arrIdx := -1;
objIdx := -1; 
IF root^.DataType = JsonDataType.JSON_DATA_OBJECT THEN 
	objIdx := 0; 
	WriteByte(SerializerConstants.START_OBJ, pDest, Offset); 
	WriteNewLine(pDest,Offset,Settings); 
	IF Settings.PrettyPrint THEN 
		Settings.IndentLevel := Settings.IndentLevel + 1; 
	END_IF
	arrObjects[objIdx] := root^.pValue;
END_IF

IF root^.DataType = JsonDataType.JSON_DATA_ARRAY THEN
	arrIdx := 0; 
	WriteByte(Value := SerializerConstants.START_ARR,pDest,Offset); 
	IF Settings.PrettyPrint THEN 
		WriteNewLine(pDest,Offset,Settings);
		Settings.IndentLevel := Settings.IndentLevel + 1; 
	END_IF
	arrArrays[arrIdx] := root^.pValue; 
END_IF
WHILE Offset < DestSize AND (objIdx >= 0 OR arrIdx >= 0) DO 
	writeIndent(pDest,Offset,Settings);
	IF ArrIdx < 0 THEN  
		pKey := arrObjects[objIdx]^.GetKeyAtIndex(curObjIdx[objIdx]);
		WriteEscapedString(pKey,pDest,Offset); 
		WriteColon(pDest,Offset,Settings); 
		pCurJsonVal := arrObjects[objIdx]^.GetValue(pKey^);
		curObjIdx[objIdx] := curObjIdx[objIdx] + 1; 
	ELSE
		arrArrays[arrIdx]^.Get(curArrIdx[arrIdx],ADR(pCurJsonVal)); 
		curArrIdx[arrIdx] := curArrIdx[arrIdx] + 1; 
	END_IF
	 
	CASE pCurJsonVal^.DataType OF 
		JSONDATATYPE.JSON_DATA_OBJECT: 
			objIdx := objIdx+1; 
			arrObjects[objIdx] := pCurJsonVal^.pValue;
			WriteByte(SerializerConstants.START_OBJ, pDest, Offset); 
			WriteNewLine(pDest,Offset,Settings); 
			IF Settings.PrettyPrint THEN 
				Settings.IndentLevel := Settings.IndentLevel + 1; 
			END_IF
		JsonDataType.JSON_DATA_ARRAY: 
			WriteByte(Value := SerializerConstants.START_ARR,pDest,Offset); 
			IF Settings.PrettyPrint THEN 
				WriteNewLine(pDest,Offset,Settings);
				Settings.IndentLevel := Settings.IndentLevel + 1; 
			END_IF
			arrIdx := arrIdx + 1; 
			arrArrays[arrIdx] := pCurJsonVal^.pValue; 
		ELSE
			SerializeJsonValue(pCurJsonVal^,pDest,Offset,Settings);
			IF arrIdx >= 0 THEN  
				IF arrArrays[arrIdx]^.Size = curArrIdx[arrIdx] THEN 
					WHILE arrArrays[arrIdx]^.Size = curArrIdx[arrIdx] DO 
						WriteNewLine(pDest,Offset,Settings); 
						Settings.IndentLevel := Settings.IndentLevel - 1; 
						WriteIndent(pDest,Offset,Settings); 
						WriteByte(Value := SerializerConstants.END_ARR,pDest,Offset);
						curArrIdx[arrIdx] := 0; 
						arrIdx := arrIdx - 1; 
						IF arrIdx < 0 THEN 
							EXIT;
						END_IF
					 END_WHILE
				ELSE
					WriteByte(SerializerConstants.COMMA,pDest,Offset);  
				END_IF
				WriteNewLine(pDest,Offset,Settings); 
			ELSE 
				WHILE arrObjects[objIdx]^.Size = curObjIdx[ObjIdx] DO
					Settings.IndentLevel := Settings.IndentLevel - 1; 
					WriteNewLine(pDest,Offset,Settings); 
					WriteIndent(pDest,Offset,Settings); 
					WriteByte(SerializerConstants.END_OBJ,pDest,Offset);
					curObjIdx[ObjIdx] := 0; 
					objIdx := objIdx - 1; 
					IF objIdx <0 THEN 
						Exit; 
					END_IF
				END_WHILE
				WriteNewLine(pDest,Offset,Settings); 
			END_IF 
			IF objIdx <0 AND arrIdx <0 THEN 
				pDest[Offset] := 0; 
				Offset := Offset + 1; 
				JsonSerializer := Offset; 	
			END_IF
	END_CASE
	
END_WHILE

END_FUNCTION

// Device/Application/Serialize/WriteByte
FUNCTION WriteByte : Bool
VAR_INPUT
    Value : BYTE;
END_VAR
VAR_IN_OUT
    pDest   : POINTER TO BYTE;
    Offset  : DINT;
END_VAR

pDest[Offset] := Value;
Offset := Offset + 1;
WriteByte := TRUE;

END_FUNCTION

// Device/Application/Serialize/WriteNewLine
FUNCTION WriteNewLine : Bool
VAR_IN_OUT
    pDest  : POINTER TO BYTE;
    Offset : DINT;
    Config : JsonSerializeConfig;
END_VAR

IF NOT Config.PrettyPrint THEN
    WriteNewline := TRUE;
    RETURN;
END_IF;

WriteByte(Value := 13, pDest := pDest, Offset := Offset);  // CR
WriteByte(Value := 10, pDest := pDest, Offset := Offset);  // LF
WriteNewline := TRUE;

END_FUNCTION

// Device/Application/Serialize/WriteIndent
FUNCTION WriteIndent : Bool
VAR_IN_OUT
    pDest  : POINTER TO BYTE;
    Offset : DINT;
    Config : JsonSerializeConfig;
END_VAR
VAR
    i          : DINT;
    TotalSpaces : DINT;
END_VAR

IF NOT Config.PrettyPrint THEN
    WriteIndent := TRUE;
    RETURN;
END_IF;

TotalSpaces := Config.IndentLevel * Config.IndentSize;
FOR i := 0 TO TotalSpaces - 1 DO
    WriteByte(Value := 32, pDest := pDest, Offset := Offset);  // space
END_FOR;

WriteIndent := TRUE;

END_FUNCTION

// Device/Application/Serialize/WriteEscapedString
FUNCTION WriteEscapedString : BOOL
VAR_INPUT
    pSource : POINTER TO BYTE;  // Null-terminated source string
END_VAR
VAR_IN_OUT
    pDest  : POINTER TO BYTE;
    Offset : DINT;
END_VAR
VAR
    CurrentChar : BYTE;
    i           : DINT;
END_VAR

// Opening quote
WriteByte(Value := 34, pDest := pDest, Offset := Offset);

i := 0;
CurrentChar := pSource[i];

WHILE CurrentChar <> 0 DO
    CASE CurrentChar OF
        34:  // " -> \"
            WriteByte(Value := 92, pDest := pDest, Offset := Offset);
            WriteByte(Value := 34, pDest := pDest, Offset := Offset);
        92:  // \ -> \\
            WriteByte(Value := 92, pDest := pDest, Offset := Offset);
            WriteByte(Value := 92, pDest := pDest, Offset := Offset);
        10:  // LF -> \n
            WriteByte(Value := 92, pDest := pDest, Offset := Offset);
            WriteByte(Value := 110, pDest := pDest, Offset := Offset);
        13:  // CR -> \r
            WriteByte(Value := 92, pDest := pDest, Offset := Offset);
            WriteByte(Value := 114, pDest := pDest, Offset := Offset);
        9:   // TAB -> \t
            WriteByte(Value := 92, pDest := pDest, Offset := Offset);
            WriteByte(Value := 116, pDest := pDest, Offset := Offset);
        8:   // BS -> \b
            WriteByte(Value := 92, pDest := pDest, Offset := Offset);
            WriteByte(Value := 98, pDest := pDest, Offset := Offset);
        12:  // FF -> \f
            WriteByte(Value := 92, pDest := pDest, Offset := Offset);
            WriteByte(Value := 102, pDest := pDest, Offset := Offset);
    ELSE
        WriteByte(Value := CurrentChar, pDest := pDest, Offset := Offset);
    END_CASE;

    i := i + 1;
    CurrentChar := pSource[i];
	END_WHILE;

// Closing quote
WriteByte(Value := 34, pDest := pDest, Offset := Offset);

WriteEscapedString := TRUE;

END_FUNCTION

// Device/Application/Serialize/WriteColon
FUNCTION WriteColon : Bool
VAR_IN_OUT
    pDest  : POINTER TO BYTE;
    Offset : DINT;
    Config : JsonSerializeConfig;
END_VAR

WriteByte(Value := 58, pDest := pDest, Offset := Offset);  // :
IF Config.PrettyPrint THEN
    WriteByte(Value := 32, pDest := pDest, Offset := Offset);  // space after colon
END_IF;

WriteColon := TRUE;

END_FUNCTION

// Device/Application/Serialize/SerializeJsonValue
FUNCTION SerializeJsonValue : BOOL
VAR_INPUT
    JsonValue : JsonType;       // The value to serialize
END_VAR
VAR_IN_OUT
    pDest  : POINTER TO BYTE;   // Destination buffer
    Offset : DINT;              // Current write position, advanced on return
    Config : JsonSerializeConfig;
END_VAR
VAR
    pBool   : POINTER TO BOOL;
    pInt    : POINTER TO DINT;
    pReal   : POINTER TO REAL;
    pString : POINTER TO BYTE;
END_VAR

CASE JsonValue.DataType OF

    JSON_DATA_NULL:
        // Write: null
        WriteByte(Value := 110, pDest := pDest, Offset := Offset);  // n
        WriteByte(Value := 117, pDest := pDest, Offset := Offset);  // u
        WriteByte(Value := 108, pDest := pDest, Offset := Offset);  // l
        WriteByte(Value := 108, pDest := pDest, Offset := Offset);  // l

    JSON_DATA_BOOL:
        pBool := JsonValue.pValue;
        IF pBool^ THEN
            // Write: true
            WriteByte(Value := 116, pDest := pDest, Offset := Offset);  // t
            WriteByte(Value := 114, pDest := pDest, Offset := Offset);  // r
            WriteByte(Value := 117, pDest := pDest, Offset := Offset);  // u
            WriteByte(Value := 101, pDest := pDest, Offset := Offset);  // e
        ELSE
            // Write: false
            WriteByte(Value := 102, pDest := pDest, Offset := Offset);  // f
            WriteByte(Value := 97,  pDest := pDest, Offset := Offset);  // a
            WriteByte(Value := 108, pDest := pDest, Offset := Offset);  // l
            WriteByte(Value := 115, pDest := pDest, Offset := Offset);  // s
            WriteByte(Value := 101, pDest := pDest, Offset := Offset);  // e
        END_IF;

    JSON_DATA_INT:
        pInt := JsonValue.pValue;
        WriteDint(Value := pInt^, pDest := pDest, Offset := Offset);

    JSON_DATA_REAL:
        pReal := JsonValue.pValue;
        WriteReal(Value := pReal^, pDest := pDest, Offset := Offset);

    JSON_DATA_STRING:
        pString := JsonValue.pValue;
        WriteEscapedString(pSource := pString, pDest := pDest, Offset := Offset);

ELSE
    SerializeJsonValue := FALSE;
    RETURN;
END_CASE;

// Null terminate
pDest[Offset] := 0;

SerializeJsonValue := TRUE;

END_FUNCTION

// Device/Application/Serialize/WriteDint
FUNCTION WriteDint : DINT
VAR_INPUT
    Value : DINT;
END_VAR
VAR_IN_OUT
    pDest  : POINTER TO BYTE;
    Offset : DINT;
END_VAR
VAR
    TempBuf  : ARRAY[0..10] OF BYTE;
    BufLen   : DINT;
    AbsValue : DINT;
    IsNeg    : BOOL;
    i        : DINT;
END_VAR

BufLen := 0;
IsNeg  := FALSE;

IF Value = 0 THEN
    WriteByte(Value := 48, pDest := pDest, Offset := Offset);  // '0'
    WriteDint := 1;
    RETURN;
END_IF;

IF Value < 0 THEN
    IsNeg    := TRUE;
    AbsValue := -Value;
ELSE
    AbsValue := Value;
END_IF;

// Extract digits in reverse order
WHILE AbsValue > 0 DO
    TempBuf[BufLen] := TO_BYTE(AbsValue MOD 10) + 48;  // digit + '0'
    AbsValue := AbsValue / 10;
    BufLen := BufLen + 1;
END_WHILE;

// Write minus sign
IF IsNeg THEN
    WriteByte(Value := 45, pDest := pDest, Offset := Offset);  // '-'
END_IF;

// Write digits in correct order (reverse the buffer)
FOR i := BufLen - 1 TO 0 BY -1 DO
    WriteByte(Value := TempBuf[i], pDest := pDest, Offset := Offset);
END_FOR;

WriteDint := BufLen;

END_FUNCTION

// Device/Application/Serialize/WriteReal
FUNCTION WriteReal : DINT
VAR_INPUT
    Value : REAL;
END_VAR
VAR_IN_OUT
    pDest  : POINTER TO BYTE;
    Offset : DINT;
END_VAR
VAR
    IntPart     : DINT;
    FracPart    : REAL;
    IsNeg       : BOOL;
    FracDigits  : DINT;
    FracBuf     : ARRAY[0..6] OF BYTE;
    i           : DINT;
    BytesWritten : DINT;
    Digit       : DINT;
END_VAR

BytesWritten := 0;
IsNeg := FALSE;

IF Value < 0.0 THEN
    IsNeg := TRUE;
    Value := -Value;
END_IF;

IntPart  := TRUNC(Value);
FracPart := Value - TO_REAL(IntPart);

// Write minus
IF IsNeg THEN
    WriteByte(Value := 45, pDest := pDest, Offset := Offset);
    BytesWritten := BytesWritten + 1;
END_IF;

// Write integer part
BytesWritten := BytesWritten + WriteDint(Value := IntPart, pDest := pDest, Offset := Offset);

// Write decimal point
WriteByte(Value := 46, pDest := pDest, Offset := Offset);  // '.'
BytesWritten := BytesWritten + 1;

// Extract fractional digits (up to 6 decimal places)
FracDigits := 0;
FOR i := 0 TO 5 DO
    FracPart := FracPart * 10.0;
    Digit := TRUNC(FracPart);
    FracBuf[i] := TO_BYTE(Digit) + 48;
    FracPart := FracPart - TO_REAL(Digit);
    FracDigits := FracDigits + 1;
END_FOR;

// Trim trailing zeros but keep at least one decimal digit
WHILE (FracDigits > 1) AND (FracBuf[FracDigits - 1] = 48) DO
    FracDigits := FracDigits - 1;
END_WHILE;

// Write fractional digits
FOR i := 0 TO FracDigits - 1 DO
    WriteByte(Value := FracBuf[i], pDest := pDest, Offset := Offset);
    BytesWritten := BytesWritten + 1;
END_FOR;

WriteReal := BytesWritten;

END_FUNCTION

// Device/Application/JsonParser2
FUNCTION_BLOCK JsonParser2
VAR_INPUT
	MAX_DOC_DEPTH : INT; 
	MAX_DOC_WIDTH : INT; 
END_VAR
VAR_OUTPUT
END_VAR
VAR
	root : JsonType;
	backingArCreatedVals : DynamicJsonTypeContainer(udSize := 1); 
	lCreatedValues : DynamicList :=(DataContainer := backingArCreatedVals); 
	backingArCreatedObj : DynamicJsonObjectContainer(udSize := 1); 
	lCreatedObj : DynamicList := (DataContainer := backingArCreatedObj); 
	backingArrayCreatedKeys : DynamicStringContainer(udSize := 1); 
	lCreatedKeys: DynamicList := (DataContainer  := backingArrayCreatedKeys); 
	strRoot : STRING := 'root';
	backingArrayArrays : DynamicJsonContainerContainer(udSize := 1);
	lCreatedLists : DynamicList := (DataContainer := backingArrayArrays); 
END_VAR

METHOD CreateJsonType : POINTER TO JSONType
VAR_INPUT
END_VAR

VAR
	_pJsonType: POINTER TO JsonType;
END_VAR
_pJsonType := __NEW(JsonType); 
lCreatedValues.PushBack(ADR(_pJsonType)); 
CreateJsonType := _pJsonType;
END_METHOD

METHOD PRIVATE DeleteJsonNode : BOOL
VAR_INPUT
	pJsonNode : POINTER TO JSONTYPE; 
END_VAR
VAR
	pString : POINTER TO STRING; 
	pLINT  : POINTER TO DINT; 
	pBOOL  : POINTER TO BOOL; 
	pFloat : POINTER TO REAL; 
	pJasonType : POINTER TO JsonType; 
	pJsonArray : POINTER TO DynamicList; 
END_VAR
IF pJsonNode = 0 THEN 
	RETURN; 
END_IF
CASE pJsonNode^.DataType OF 
	JSON_DATA_NULL: 
// nothing to clean	
    JSON_DATA_BOOL: 
		pBool := pJsonNode^.pValue; 
		__DELETE(pBool);
    JSON_DATA_INT:
		pLINT := pJsonNode^.pValue;
		__DELETE(pLINT); 
    JSON_DATA_REAL: 
		pFloat := pJsonNode^.pValue; 
		__DELETE(pFloat);
    JSON_DATA_STRING: 
		pString :=pJsonNode^.pValue;
		__DELETE(pString); 
	JSON_DATA_ARRAY:
		pJsonArray := pJsonNode^.pValue; 
		__DELETE(pJsonArray); 
END_CASE
	__DELETE(pJsonNode);
END_METHOD

//FB_Exit must be implemented explicitly. If there is an implementation, then the
//method is called before the controller removes the code of the function block instance
//(implicit call). The return value is not evaluated.
METHOD  FB_Exit: BOOL
VAR_INPUT
    bInCopyCode: BOOL;  // TRUE: the exit method is called in order to leave the instance which will be copied afterwards (online change).  
END_VAR
This^.Clean();
END_METHOD

METHOD GetRootDoc : POINTER TO JsonType; 
VAR_INPUT
END_VAR
VAR
	pJson : POINTER TO JsonObjectManager; 
	pJsonType : POINTER TO JsonType; 
END_VAR
pJson := root.pValue; 
IF pJSON = 0 THEN 
	RETURN; 
END_IF
pJsonType := pJson^.GetValue('root');
GetRootDoc := pJsonType;
END_METHOD

METHOD Parse : BOOL
VAR_INPUT
	pJsonStr : POINTER TO BYTE; 
	StrSize  : LINT; 
END_VAR
VAR
	Offset : LINT; 
	stJsonToken: JsonToken;
	arrObjects : ARRAY[0..Parameters.MAX_DOC_DEPTH] OF POINTER TO JsonObjectManager; 
	arrArrays  : ARRAY[0..Parameters.MAX_DOC_DEPTH] OF POINTER TO DynamicList; 
	objIdx : INT; 
	arrIdx : INT; 
	bArr : BOOL; 
	bArObj : BOOL; 
	pBool: POINTER TO BOOL;
	bNeedKey : BOOL; 
	HasDecimal: BOOL;
	jsonNodeVal: JsonType;
	pJsonObj: POINTER TO JSONObject;
	pJsonArray: POINTER TO DynamicList;
	pJsonType: POINTER TO JSONType;
	bFirstObj: BOOL;
	pRootOBJ: POINTER TO JsonObjectManager;
	strKey : POINTER TO BYTE;  
END_VAR
PARSE := FALSE; 
THIS^.Clean(); 
Offset := 0; 
objIdx := 0; 
arrIdx := -1; 
THIS^.root.DataType := JsonDataType.JSON_DATA_OBJECT;
pRootOBJ := CreateObj();  
THIS^.root.pValue := pRootObj; 
arrObjects[0] := pRootObj; 
bArr := FALSE; 
bNeedKey := TRUE; 
bFirstObj := TRUE; 
strKey := ADR(strRoot); 
WHILE Offset < StrSize DO 
	stJsonToken := GetNextJsonToken(pJsonStr,StrSize, Offset := Offset); 
	CASE stJsonToken.TokenType OF 
		JSON_TOKEN_NULL, JSON_TOKEN_TRUE, JSON_TOKEN_FALSE, JSON_TOKEN_NUMBER:
			jsonNodeVal := JsonHadlr(pJsonStr,stJsonToken);
			IF bARR AND NOT bARObj THEN 
				pJsonType := CreateJsonType(); 
				pJsonType^:=jsonNodeVal; 
				arrArrays[arrIdx]^.PushBack(ADR(pJsonType)); 
			ELSE 
				pJsonType := CreateJsonType(); 
				pJsonType^:=jsonNodeVal; 
				arrObjects[objIdx]^.Put(strKey, pJsonType); 
				bNeedKey := TRUE;  
			END_IF
		JSON_TOKEN_STRING: 
			jsonNodeVal := JsonHadlr(pJsonStr,stJsonToken);
			IF bNeedKey THEN 
				strKey := jsonNodeVal.pValue; 
				lCreatedKeys.PushBack(ADR(strKey)); 
				bNeedKey := FALSE; 
			ELSIF bArr THEN 
				pJsonType := CreateJsonType(); 
				pJsonType^:=jsonNodeVal; 
				arrArrays[arrIdx]^.PushBack(ADR(pJsonType));  
			ELSE
				pJsonType := CreateJsonType(); 
				pJsonType^:=jsonNodeVal; 
				arrObjects[objIdx]^.Put(strKey, pJsonType); 
				bNeedKey := TRUE; 
			END_IF
    	JSON_TOKEN_LBRACE:      // {
			pJsonObj := CreateObj(); 
			pJsonType := CreateJsonType(); 
			pJsonType^.pValue := pJsonObj; 
			pJsonType^.DataType :=JsonDataType.JSON_DATA_OBJECT;  
			IF bARR THEN 
				arrArrays[arrIdx]^.PushBack(ADR(pJsonType)); 
				bArObj := TRUE; 
			ELSE
				arrObjects[objIdx]^.Put(strKey,pJsonType); 
			END_IF
			
			objIdx := objIdx + 1; 
			arrObjects[objIdx] := pJsonObj;
			bNeedKey := TRUE;  
			
    	JSON_TOKEN_RBRACE:      // }
			objIdx := objIdx - 1; 
			bArObj := FALSE; 
			
    	JSON_TOKEN_LBRACKET:    // [
			pJsonArray := CreateArray(); 
			arrIdx := arrIdx + 1; 
			arrArrays[arrIdx] := pJsonArray; 
			pJsonType := CreateJsonType(); 
			pJsonType^.DataType := JsonDataType.JSON_DATA_ARRAY; 
			pJsonType^.pValue := pJsonArray; 
			IF bArr THEN 
				arrArrays[arrIdx-1]^.PushBack(ADR(pJsonType)); 
			ELSE
				arrObjects[objIdx]^.Put(strKey, pJsonType); 
			END_IF
			bArr := TRUE; 
			bNeedKey := FALSE; 
			
    	JSON_TOKEN_RBRACKET:    // ]
			arrIdx := arrIdx - 1; 
			IF arrIdx < 0 THEN 
				bArr := FALSE;
				bNeedKey := TRUE; 
			END_IF
			 
			
    	JSON_TOKEN_COMMA:       // ,
		
    	JSON_TOKEN_COLON:       // :
		
    	JSON_TOKEN_EOF:
		IF arrIdx = -1 AND objIdx = 0 THEN 
			Parse := TRUE;
		ELSE
			Clean();
			root.pValue := 0; 
		END_IF
			EXIT; 
    	JSON_TOKEN_ERROR: 
			EXIT; 
	END_CASE
END_WHILE
END_METHOD

METHOD Clean : BOOL
VAR_INPUT
	
END_VAR
VAR 
	arrIdx : INT;  
	pJsonData: POINTER TO JsonTYPE;
	pJsonManager: Pointer TO JsonObjectManager;
	pString: POINTER TO BYTE;
	pBackingLists : Pointer TO DynamicJsonTypeContainer;
END_VAR
arrIdx := 0; 
WHILE lCreatedValues.GetIterator().Next(ADR(pJsonData)) DO 
	IF pJsonData <> 0 THEN 
		DeleteJsonNode(pJsonData); 
	END_IF
	pJsonData := 0; 
END_WHILE
WHILE lCreatedKeys.GetIterator().Next(ADR(pString)) DO 
	IF pString <> 0 THEN
		__DELETE(pString);
	END_IF 
	pString := 0;  
END_WHILE
WHILE lCreatedObj.GetIterator().Next(ADR(pJsonManager)) DO
	pJsonManager^.Destroy(); 
	__DELETE(pJsonManager); 
END_WHILE
WHILE lCreatedLists.GetIterator().Next(ADR(pBackingLists)) DO 
	__DELETE(pBackingLists); 
END_WHILE
lCreatedValues.Clear(); 
lCreatedObj.Clear(); 
lCreatedKeys.Clear(); 
lCreatedLists.Clear();
END_METHOD

METHOD PRIVATE CreateArray : POINTER TO DynamicList
VAR_INPUT
END_VAR

VAR
	_pBacking: POINTER TO DynamicJsonTypeContainer;
	_lArray: POINTER TO DynamicList;
END_VAR
_pBacking := __NEW(DynamicJsonTypeContainer(udSize := 1)); 
lCreatedLists.PushBack(ADR(_pBacking)); 
_lArray := __NEW(DynamicList); 
_lArray^(DataContainer := _pBacking^); 
CreateArray := _lArray;
END_METHOD

METHOD CreateObj : Pointer TO JsonObjectManager
VAR_INPUT
END_VAR

VAR
	pJsonManager: POINTER TO JsonObjectManager;
END_VAR
pJsonManager := __NEW(JsonObjectManager); 
pJsonManager^.Create(); 
lCreatedObj.PushBack(ADR(pJsonManager));
CreateObj := pJsonManager;
END_METHOD

END_FUNCTION_BLOCK

// Device/Application/ResizableMem (Not Fully Tested)/DynamicJsonObjectContainer
{attribute 'enable_dynamic_creation'}
FUNCTION_BLOCK DynamicJsonObjectContainer IMPLEMENTS iDynamicDataContainer
VAR_INPUT
	udSize : UDINT; 
END_VAR
VAR_OUTPUT
END_VAR
VAR
	_ptrBackingArray : POINTER TO POINTER TO JsonObjectManager;
	_ptrTempNewArray : POINTER TO POINTER TO JsonObjectManager;  
	_size : UDINT; 
	_tData : POINTER TO JsonObjectManager; 
	_pData : POINTER TO POINTER TO jsonObjectManager; 
	_newSize: UDINT;
	_byteSize : UDINT; 
END_VAR

_byteSize := SIZEOF(_tData); 
_newSize := udSize * _byteSize;
_ptrBackingArray := __NEW(BYTE,_newSize); 
_size := udSize;

METHOD CopyToNew : BOOL
VAR_INPUT
	indexOld	: UDINT;
	indexNew	: UDINT;
END_VAR
CopyToNew := FALSE; 
IF indexOld < _size/2 AND indexNew < _size THEN 
	_ptrTempNewArray[indexNew] := _ptrBackingArray[indexOld]; 
	CopyToNew := TRUE; 
END_IF
END_METHOD

//FB_Exit must be implemented explicitly. If there is an implementation, then the
//method is called before the controller removes the code of the function block instance
//(implicit call). The return value is not evaluated.
METHOD FB_Exit: BOOL
VAR_INPUT
    bInCopyCode: BOOL;  // TRUE: the exit method is called in order to leave the instance which will be copied afterwards (online change).  
END_VAR
VAR
	i: UDINT;
END_VAR
IF _ptrBackingArray <> 0 THEN 
	__DELETE(_ptrBackingArray); 
END_IF
IF _ptrTempNewArray <> 0 THEN 
	__DELETE(_ptrTempNewArray); 
END_IF
END_METHOD

METHOD Get : BOOL
VAR_INPUT
	index	: UDINT;
	pData	: PVoid;
END_VAR
IF index < _size THEN 
	_pData := pData; 
	_pData^ := _ptrBackingArray[index]; 
	GET := TRUE; 
ELSE 
	GET := FALSE; 
END_IF
END_METHOD

METHOD GetNew : BOOL
VAR_INPUT
	index	: UDINT;
	pData	: PVoid;
END_VAR
IF _ptrTempNewArray <> 0 AND index < _size THEN 
	_pData := pData; 
	_pData^ :=_ptrTempNewArray[index]; 
	GetNew := TRUE; 
ELSE 
	GetNew := FALSE; 
END_IF
END_METHOD

METHOD GetNewPointer : PVoid
VAR_INPUT
	index	: UDINT;
END_VAR
IF _ptrTempNewArray <> 0 AND index < _size THEN 
	GetNewPointer := ADR(_ptrTempNewArray[index]); 
ELSE 
	GetNewPointer := 0; 
END_IF
END_METHOD

METHOD GetPointer : PVoid
VAR_INPUT
	index	: UDINT;
END_VAR
IF index < _size THEN 
	GetPointer := ADR(_ptrBackingArray[index]); 
ELSE 
	GetPointer := 0; 
END_IF
END_METHOD

METHOD Put : BOOL
VAR_INPUT
	index	: UDINT;
	pData	: PVoid;
END_VAR
_pData := pData; 
Put := FALSE; 
IF index < _size THEN 
	_ptrBackingArray[index] := _pData^; 
	Put := TRUE; 
END_IF
END_METHOD

METHOD EndResize : BOOL
__DELETE(_ptrBackingArray); 
_ptrBackingArray := _ptrTempNewArray; 
_ptrTempNewArray := 0;
END_METHOD

//FB_Init is always available implicitly and it is used primarily for initialization.
//The return value is not evaluated. For a specific influence, you can also declare the
//methods explicitly and provide additional code there with the standard initialization
//code. You can evaluate the return value.
METHOD FB_Init: BOOL
VAR_INPUT
    bInitRetains: BOOL; // TRUE: the retain variables are initialized (reset warm / reset cold)
    bInCopyCode: BOOL;  // TRUE: the instance will be copied to the copy code afterward (online change) 
	udSize      : UDINT;   
END_VAR
this^(udSize := udSize);
END_METHOD

METHOD GetSize : UDINT
GetSize :=_size;
END_METHOD

METHOD StartResize : BOOL
VAR
	_newSize: UDINT;
END_VAR
_newSize := (2* _size)*_byteSize;
_ptrTempNewArray := __NEW(BYTE,_newSize); 
_size := _size * 2;
END_METHOD

END_FUNCTION_BLOCK

// Device/Application/ResizableMem (Not Fully Tested)/DynamicJsonContainerContainer
{attribute 'enable_dynamic_creation'}
FUNCTION_BLOCK DynamicJsonContainerContainer IMPLEMENTS iDynamicDataContainer
VAR_INPUT
	udSize : UDINT; 
END_VAR
VAR_OUTPUT
END_VAR
VAR
	_ptrBackingArray : POINTER TO POINTER TO DynamicJsonTypeContainer;
	_ptrTempNewArray : POINTER TO POINTER TO DynamicJsonTypeContainer;  
	_size : UDINT; 
	_tData : POINTER TO DynamicJsonTypeContainer; 
	_pData : POINTER TO POINTER TO DynamicJsonTypeContainer; 
	_newSize: UDINT;
	_byteSize : UDINT; 
END_VAR

_byteSize := SIZEOF(_tData); 
_newSize := udSize * _byteSize;
_ptrBackingArray := __NEW(BYTE,_newSize); 
_size := udSize;

METHOD CopyToNew : BOOL
VAR_INPUT
	indexOld	: UDINT;
	indexNew	: UDINT;
END_VAR
CopyToNew := FALSE; 
IF indexOld < _size/2 AND indexNew < _size THEN 
	_ptrTempNewArray[indexNew] := _ptrBackingArray[indexOld]; 
	CopyToNew := TRUE; 
END_IF
END_METHOD

METHOD EndResize : BOOL
__DELETE(_ptrBackingArray); 
_ptrBackingArray := _ptrTempNewArray; 
_ptrTempNewArray := 0;
END_METHOD

//FB_Exit must be implemented explicitly. If there is an implementation, then the
//method is called before the controller removes the code of the function block instance
//(implicit call). The return value is not evaluated.
METHOD FB_Exit: BOOL
VAR_INPUT
    bInCopyCode: BOOL;  // TRUE: the exit method is called in order to leave the instance which will be copied afterwards (online change).  
END_VAR
VAR
	i: UDINT;
END_VAR
IF _ptrBackingArray <> 0 THEN 
	__DELETE(_ptrBackingArray); 
END_IF
IF _ptrTempNewArray <> 0 THEN 
	__DELETE(_ptrTempNewArray); 
END_IF
END_METHOD

METHOD Get : BOOL
VAR_INPUT
	index	: UDINT;
	pData	: PVoid;
END_VAR
IF index < _size THEN 
	_pData := pData; 
	_pData^ := _ptrBackingArray[index]; 
	GET := TRUE; 
ELSE 
	GET := FALSE; 
END_IF
END_METHOD

METHOD GetNew : BOOL
VAR_INPUT
	index	: UDINT;
	pData	: PVoid;
END_VAR
IF _ptrTempNewArray <> 0 AND index < _size THEN 
	_pData := pData; 
	_pData^ :=_ptrTempNewArray[index]; 
	GetNew := TRUE; 
ELSE 
	GetNew := FALSE; 
END_IF
END_METHOD

METHOD GetNewPointer : PVoid
VAR_INPUT
	index	: UDINT;
END_VAR
IF _ptrTempNewArray <> 0 AND index < _size THEN 
	GetNewPointer := ADR(_ptrTempNewArray[index]); 
ELSE 
	GetNewPointer := 0; 
END_IF
END_METHOD

METHOD GetPointer : PVoid
VAR_INPUT
	index	: UDINT;
END_VAR
IF index < _size THEN 
	GetPointer := ADR(_ptrBackingArray[index]); 
ELSE 
	GetPointer := 0; 
END_IF
END_METHOD

METHOD GetSize : UDINT
GetSize :=_size;
END_METHOD

METHOD Put : BOOL
VAR_INPUT
	index	: UDINT;
	pData	: PVoid;
END_VAR
_pData := pData; 
Put := FALSE; 
IF index < _size THEN 
	_ptrBackingArray[index] := _pData^; 
	Put := TRUE; 
END_IF
END_METHOD

//FB_Init is always available implicitly and it is used primarily for initialization.
//The return value is not evaluated. For a specific influence, you can also declare the
//methods explicitly and provide additional code there with the standard initialization
//code. You can evaluate the return value.
METHOD FB_Init: BOOL
VAR_INPUT
    bInitRetains: BOOL; // TRUE: the retain variables are initialized (reset warm / reset cold)
    bInCopyCode: BOOL;  // TRUE: the instance will be copied to the copy code afterward (online change) 
	udSize      : UDINT;   
END_VAR
this^(udSize := udSize);
END_METHOD

METHOD StartResize : BOOL
VAR
	_newSize: UDINT;
END_VAR
_newSize := (2* _size)*_byteSize;
_ptrTempNewArray := __NEW(BYTE,_newSize); 
_size := _size * 2;
END_METHOD

END_FUNCTION_BLOCK

// Device/Application/GetNextJsonToken
FUNCTION GetNextJsonToken : JsonToken
VAR_INPUT
	JsonString : POINTER TO BYTE; 
	StrSize    : LINT; 
END_VAR
VAR_IN_OUT
	Offset : LINT;
END_VAR
VAR
	Token : JsonToken;
    CurrentChar : BYTE;
    StartOffset : LINT;
    i : DINT;
    IsValid : BOOL;
END_VAR

Token.TokenType := JSON_TOKEN_ERROR;
Token.StartIndex := 0;
Token.Length := 0;

// Skip whitespace
WHILE (Offset <= StrSize) DO
    CurrentChar := JsonString[Offset]; 
    IF CurrentChar = 32 OR CurrentChar = 9 OR CurrentChar = 10 OR CurrentChar = 13 THEN // space, tab, LF, CR
        Offset := Offset + 1;
    ELSE
        EXIT;
    END_IF;
END_WHILE;

// Check for end of string
IF Offset > StrSize THEN
    Token.TokenType := JSON_TOKEN_EOF;
    Token.StartIndex := Offset;
    GetNextJsonToken := Token;
    RETURN;
END_IF;

Token.StartIndex := Offset;
CurrentChar := JsonString[Offset]; 

// Single character tokens
CASE CurrentChar OF
    123: // {
        Token.TokenType := JSON_TOKEN_LBRACE;
        Token.Length := 1;
        Offset := Offset + 1;
        GetNextJsonToken := Token;
        RETURN;
        
    125: // }
        Token.TokenType := JSON_TOKEN_RBRACE;
        Token.Length := 1;
        Offset := Offset + 1;
        GetNextJsonToken := Token;
        RETURN;
        
    91: // [
        Token.TokenType := JSON_TOKEN_LBRACKET;
        Token.Length := 1;
        Offset := Offset + 1;
        GetNextJsonToken := Token;
        RETURN;
        
    93: // ]
        Token.TokenType := JSON_TOKEN_RBRACKET;
        Token.Length := 1;
        Offset := Offset + 1;
        GetNextJsonToken := Token;
        RETURN;
        
    44: // ,
        Token.TokenType := JSON_TOKEN_COMMA;
        Token.Length := 1;
        Offset := Offset + 1;
        GetNextJsonToken := Token;
        RETURN;
        
    58: // :
        Token.TokenType := JSON_TOKEN_COLON;
        Token.Length := 1;
        Offset := Offset + 1;
        GetNextJsonToken := Token;
        RETURN;
        
    34: // " (string)
        Offset := Offset + 1;
        WHILE Offset <= StrSize DO
            CurrentChar := JsonString[Offset];
            IF CurrentChar = 92 THEN // backslash (escape)
                Offset := Offset + 2; // Skip escape and next char
            ELSIF CurrentChar = 34 THEN // closing quote
                Offset := Offset + 1;
                Token.TokenType := JSON_TOKEN_STRING;
                Token.Length := TO_DINT(Offset - Token.StartIndex);
                GetNextJsonToken := Token;
                RETURN;
            ELSE
                Offset := Offset + 1;
            END_IF;
        END_WHILE;
        Token.TokenType := JSON_TOKEN_ERROR;
        GetNextJsonToken := Token;
        RETURN;
	0://String TERM 
		Token.TokenType := JsonTokenType.JSON_TOKEN_EOF; 
		Token.Length := 0; 
		Token.StartIndex := Offset; 
		GetNextJsonToken := Token; 
		RETURN; 
END_CASE;

// Check for number (starts with - or digit)
IF (CurrentChar = 45) OR (CurrentChar >= 48 AND CurrentChar <= 57) THEN // - or 0-9
    StartOffset := Offset;
    
    // Skip minus sign
    IF CurrentChar = 45 THEN
        Offset := Offset + 1;
    END_IF;
    
    // Integer part
    WHILE Offset <= StrSize DO
        CurrentChar := JsonString[Offset];
        IF CurrentChar >= 48 AND CurrentChar <= 57 THEN // 0-9
            Offset := Offset + 1;
        ELSE
            EXIT;
        END_IF;
    END_WHILE;
    
    // Decimal part
    IF Offset <= StrSize AND JsonString[Offset] = 46 THEN // .
        Offset := Offset + 1;
        WHILE Offset <= StrSize DO
            CurrentChar := JsonString[Offset];
            IF CurrentChar >= 48 AND CurrentChar <= 57 THEN
                Offset := Offset + 1;
            ELSE
                EXIT;
            END_IF;
        END_WHILE;
    END_IF;
    
    // Exponent part
    IF Offset <= StrSize THEN
        CurrentChar := JsonString[Offset];
        IF CurrentChar = 101 OR CurrentChar = 69 THEN // e or E
            Offset := Offset + 1;
            IF Offset <= StrSize THEN
                CurrentChar := JsonString[Offset];
                IF CurrentChar = 43 OR CurrentChar = 45 THEN // + or -
                    Offset := Offset + 1;
                END_IF;
            END_IF;
            WHILE Offset <= StrSize DO
                CurrentChar := JsonString[Offset];
                IF CurrentChar >= 48 AND CurrentChar <= 57 THEN
                    Offset := Offset + 1;
                ELSE
                    EXIT;
                END_IF;
            END_WHILE;
        END_IF;
    END_IF;
    
    Token.TokenType := JSON_TOKEN_NUMBER;
    Token.Length := TO_DINT(Offset - Token.StartIndex);
    GetNextJsonToken := Token;
    RETURN;
END_IF;

// Check for keywords: null, true, false
IF GetSubString(JsonString,StrSize,4,Offset) = 'null' THEN
    Token.TokenType := JSON_TOKEN_NULL;
    Token.Length := 4;
    Offset := Offset + 4;
    GetNextJsonToken := Token;
    RETURN;
END_IF;

IF GetSubString(JsonString,StrSize,4,Offset) = 'true' THEN
    Token.TokenType := JSON_TOKEN_TRUE;
    Token.Length := 4;
    Offset := Offset + 4;
    GetNextJsonToken := Token;
    RETURN;
END_IF;

IF GetSubString(JsonString,StrSize,5,Offset) = 'false' THEN
    Token.TokenType := JSON_TOKEN_FALSE;
    Token.Length := 5;
    Offset := Offset + 5;
    GetNextJsonToken := Token;
    RETURN;
END_IF;

// If we get here, it's an error
Token.TokenType := JSON_TOKEN_ERROR;
GetNextJsonToken := Token;

END_FUNCTION

// Device/Application/GetSubString
FUNCTION GetSubString : String
VAR_INPUT
	StrPtr  : POINTER TO BYTE; 
	StrLen  : LINT; 
	SubStringLen : INT; 
	SubStringStart : LINT; 
END_VAR
VAR
	_i: LINT;
END_VAR

GetSubString :=''; 
IF SubStringStart + SubStringLen > StrLen THEN 
	RETURN; 
END_IF
IF subStringLen <1 THEN 
	RETURN; 
END_IF
FOR _i := SubStringStart TO SubStringStart + subStringLen-1 DO 
	GetSubString[_i - SubStringStart] := StrPtr[_i]; 
END_FOR
GetSubString[_i - SubStringStart] := 0;

END_FUNCTION

// Device/Application/JsonHadlr
FUNCTION JsonHadlr : JsonType
VAR_INPUT
	pJsonString : POINTER TO BYTE;  // Pointer to JSON string bytes
    Token : JsonToken;              // Token to parse
END_VAR
VAR
	Result : JsonType;
    pTokenStart : POINTER TO BYTE;
    pReal : POINTER TO REAL;
    pInt : POINTER TO DINT;
    pBool : POINTER TO BOOL;
    pString : POINTER TO BYTE;
    i : DINT;
    CurrentChar : BYTE;
    StringLen : DINT;
    IsNegative : BOOL;
    IntValue : DINT;
    RealValue : REAL;
    DecimalPart : REAL;
    DecimalDivisor : REAL;
    HasDecimal : BOOL;
    TempChar : BYTE;
	StrLenVal: DINT;
	j : LINT; 
END_VAR

// Initialize result
Result.DataType := JSON_DATA_NULL;
Result.pValue := 0;

// Get pointer to start of token
pTokenStart := pJsonString + TO_LWORD(Token.StartIndex);

// Parse based on token type
CASE Token.TokenType OF
    
    JSON_TOKEN_NULL:
        Result.DataType := JSON_DATA_NULL;
        Result.pValue := 0;
    
    JSON_TOKEN_TRUE, JSON_TOKEN_FALSE:
        // Allocate memory for boolean
        pBool := __NEW(BOOL);
        IF pBool <> 0 THEN
            IF Token.TokenType = JSON_TOKEN_TRUE THEN
                pBool^ := TRUE;
            ELSE
                pBool^ := FALSE;
            END_IF;
            Result.DataType := JSON_DATA_BOOL;
            Result.pValue := pBool;
        END_IF;
    
    JSON_TOKEN_NUMBER:
        // Check if number has decimal point or exponent
        HasDecimal := FALSE;
        FOR i := 0 TO Token.Length - 1 DO
            CurrentChar := pTokenStart[i];
            IF (CurrentChar = 46) OR (CurrentChar = 101) OR (CurrentChar = 69) THEN // . e E
                HasDecimal := TRUE;
                EXIT;
            END_IF;
        END_FOR;
        
        IF HasDecimal THEN
            // Parse as REAL
            pReal := __NEW(REAL);
            IF pReal <> 0 THEN
                RealValue := 0.0;
                IsNegative := FALSE;
                i := 0;
                
                // Check for negative sign
                CurrentChar := pTokenStart[i];
                IF CurrentChar = 45 THEN  // -
                    IsNegative := TRUE;
                    i := i + 1;
                END_IF;
                
                // Parse integer part
                WHILE i < Token.Length DO
                    CurrentChar := pTokenStart[i];
                    IF (CurrentChar >= 48) AND (CurrentChar <= 57) THEN  // 0-9
                        RealValue := RealValue * 10.0 + TO_REAL(CurrentChar - 48);
                        i := i + 1;
                    ELSE
                        EXIT;
                    END_IF;
                END_WHILE;
                
                // Parse decimal part if present
                IF (i < Token.Length) AND (pTokenStart[i] = 46) THEN  // .
                    i := i + 1;
                    DecimalPart := 0.0;
                    DecimalDivisor := 10.0;
                    
                    WHILE i < Token.Length DO
                        CurrentChar := pTokenStart[i];
                        IF (CurrentChar >= 48) AND (CurrentChar <= 57) THEN
                            DecimalPart := DecimalPart + TO_REAL(CurrentChar - 48) / DecimalDivisor;
                            DecimalDivisor := DecimalDivisor * 10.0;
                            i := i + 1;
                        ELSE
                            EXIT;
                        END_IF;
                    END_WHILE;
                    
                    RealValue := RealValue + DecimalPart;
                END_IF;
                
                // Note: Exponent parsing omitted for brevity, add if needed
                
                IF IsNegative THEN
                    RealValue := -RealValue;
                END_IF;
                
                pReal^ := RealValue;
                Result.DataType := JSON_DATA_REAL;
                Result.pValue := pReal;
            END_IF;
        ELSE
            // Parse as integer (DINT)
            pInt := __NEW(DINT);
            IF pInt <> 0 THEN
                IntValue := 0;
                IsNegative := FALSE;
                i := 0;
                
                // Check for negative sign
                CurrentChar := pTokenStart[i];
                IF CurrentChar = 45 THEN  // -
                    IsNegative := TRUE;
                    i := i + 1;
                END_IF;
                
                // Parse digits
                WHILE i < Token.Length DO
                    CurrentChar := pTokenStart[i];
                    IF (CurrentChar >= 48) AND (CurrentChar <= 57) THEN  // 0-9
                        IntValue := IntValue * 10 + TO_DINT(CurrentChar - 48);
                        i := i + 1;
                    ELSE
                        EXIT;
                    END_IF;
                END_WHILE;
                
                IF IsNegative THEN
                    IntValue := -IntValue;
                END_IF;
                
                pInt^ := IntValue;
                Result.DataType := JSON_DATA_INT;
                Result.pValue := pInt;
            END_IF;
        END_IF;
    
    JSON_TOKEN_STRING:
		// Allocate memory for string (length + 1 for null terminator)
		StringLen := Token.Length; 
		StrLenVal := StringLen - 1; 
        pString := __NEW(BYTE, StrLenVal);
		j := 0; 
        IF pString <> 0 THEN
            FOR i :=1 TO StringLen -2 DO//Skip the " 
                CurrentChar := pTokenStart[i];
                // Handle escape sequences
                IF CurrentChar = 92 THEN  // \ (backslash)
					i := i + 1; 
                    TempChar := pTokenStart[i];
                    CASE TempChar OF
                        110: pString[j] := 10;  // \n -> LF
                        116: pString[j] := 9;   // \t -> TAB
                        114: pString[j] := 13;  // \r -> CR
                        34:  pString[j] := 34;  // \" -> "
                        92:  pString[j] := 92;  // \\ -> \
                    ELSE
                        pString[j] := TempChar;
                    END_CASE;
                ELSE
                    pString[j] := CurrentChar;  // Adjust for escape handling
                END_IF;
				j := j + 1; 
            END_FOR;
            
            // Add null terminator
            pString[j] := 0;
            
            Result.DataType := JSON_DATA_STRING;
            Result.pValue := pString;
        END_IF;
    
ELSE
    Result.DataType := JSON_DATA_NULL;
    Result.pValue := 0;
END_CASE;

JsonHadlr := Result;

END_FUNCTION

// Device/Application/JsonSaxWriter
{attribute 'hide_all_locals'}
FUNCTION_BLOCK JsonSaxWriter
VAR_INPUT
END_VAR
VAR_OUTPUT
	initStatus: POINTER TO JsonType;
END_VAR
VAR
	_arrObjects : ARRAY[0..Parameters.MAX_DOC_DEPTH] OF POINTER TO JsonObjectManager; 
	_arrArrays  : ARRAY[0..Parameters.MAX_DOC_DEPTH] OF POINTER TO DynamicList; 
	_objIdx : INT; 
	_arrIdx : INT; 
	_curArrIdx : ARRAY[0.. Parameters.MAX_DOC_DEPTH] OF UDINT;  
	_bArr : BOOL; 
	_Key  : POINTER TO BYTE; 
	_root : JsonType;
	_backingArCreatedVals : DynamicJsonTypeContainer(udSize := 1); 
	_lCreatedValues : DynamicList :=(DataContainer := _backingArCreatedVals); 
	_backingArCreatedObj : DynamicJsonObjectContainer(udSize := 1); 
	_lCreatedObj : DynamicList := (DataContainer := _backingArCreatedObj); 
	_backingArrayCreatedKeys : DynamicStringContainer(udSize := 1); 
	_lCreatedKeys: DynamicList := (DataContainer  := _backingArrayCreatedKeys);
	backingArrayArrays : DynamicJsonContainerContainer(udSize := 1);
	lCreatedLists : DynamicList := (DataContainer := backingArrayArrays);  
	_strRoot : STRING := 'root';
	_bInit : BOOL; 
	_AddKey: BOOL;
	_bRootAdded : BOOL; 
END_VAR

METHOD AddBool : BOOL
VAR_INPUT
  value : BOOL;
END_VAR
VAR
	pJsonType: POINTER TO JSONType;
	pBool: POINTER TO BOOL;
END_VAR
IF NOT _bInit AND NOT _barr AND NOT _AddKey THEN
	AddBool := FALSE; 
	RETURN; 
END_IF
pJsonType := CreateJsonType(); 
pJsonType^.DataType := JsonDataType.JSON_DATA_BOOL; 
pBool := __NEW(BOOL); 
pBool^ := value;
pJsonType^.pValue := pBool;  
IF NOT _bArr THEN 
	_arrObjects[_ObjIdx]^.Put(_key,pJsonType); 
  	_AddKey := FALSE; 
ELSE 
	_arrArrays[_arrIdx]^.PushBack(ADR(pJsonType)); 
END_IF
END_METHOD

METHOD AddChild : BOOL
VAR_INPUT
	value : POINTER TO JsonType; 
END_VAR
IF NOT _bInit AND NOT _barr AND NOT _AddKey THEN 
	RETURN; 
END_IF
IF NOT _bArr THEN 
	_arrObjects[_objIdx]^.Put(_key,value); 
	_AddKey := FALSE; 
ELSE 
	_arrArrays[_arrIdx]^.PushBack(ADR(value)); 
END_IF
END_METHOD

METHOD AddDint : BOOL
VAR_INPUT
  value : DINT;
END_VAR

VAR
	pJson : POINTER TO JsonType;
	pDint: POINTER TO DINT;
END_VAR
IF NOT _bInit AND NOT _barr AND NOT _AddKey THEN 
	RETURN; 
END_IF
pJson := CreateJsonType(); 
pJson^.DataType := JSONDATATYPE.JSON_DATA_INT; 
pDint := __NEW(DINT); 
pDint^ := value;
pJson^.pValue := pDint; 
IF NOT _bArr THEN 
	_arrObjects[_objIdx]^.Put(_key,pJson); 
	_AddKey := FALSE; 
ELSE 
	_arrArrays[_arrIdx]^.PushBack(ADR(pJson)); 
END_IF
END_METHOD

METHOD AddFloat : BOOL
VAR_INPUT
	value : REAL; 
END_VAR
VAR
	pJson: POINTER TO JsonType;
	pReal : POINTER TO REAL; 
END_VAR
IF NOT _bInit AND NOT _barr AND NOT _AddKey THEN 
	RETURN; 
END_IF
pJson := CreateJsonType(); 
pJson^.DataType := JSONDATATYPE.JSON_DATA_REAL; 
pReal := __NEW(REAL); 
pReal^ := value;
pJson^.pValue := pReal; 
IF NOT _bArr THEN 
	_arrObjects[_objIdx]^.Put(_key,pJson); 
	_AddKey := FALSE; 
ELSE 
	_arrArrays[_arrIdx]^.PushBack(ADR(pJson)); 
END_IF
END_METHOD

METHOD AddKey : BOOL
VAR_IN_OUT CONSTANT
	key: STRING;
END_VAR

VAR

	_i: DINT;
END_VAR
_i := 0; 
WHILE Key[_i] <> 0 DO
	_i := _i + 1; 
END_WHILE
_i := _i + 1; 
_key := __NEW(BYTE,_i); 
_i := 0; 
WHILE Key[_i] <> 0 DO
	_key[_i] := key[_i]; 
	_i := _i + 1; 
END_WHILE
_key[_i] := 0; 
_lCreatedKeys.PushBack(ADR(_key)); 
_AddKey := TRUE; 
AddKey := TRUE;
END_METHOD

METHOD AddNull 
VAR_INPUT
END_VAR

VAR
	pJson: Pointer TO JsonTYpe;
END_VAR
IF NOT _bInit AND NOT _barr AND NOT _AddKey THEN 
	RETURN; 
END_IF
pJson := CreateJsonType(); 
pJson^.DataType := JSONDATATYPE.JSON_DATA_NULL; 
pJson^.pValue := 0; 
IF NOT _bArr THEN 
	_arrObjects[_objIdx]^.Put(_key,pJson); 
	_AddKey := FALSE; 
ELSE 
	_arrArrays[_arrIdx]^.PushBack(ADR(pJson)); 
END_IF
_AddKey := FALSE;
END_METHOD

METHOD AddString : BOOL
VAR_IN_OUT CONSTANT
	value: STRING;
END_VAR
VAR
	pJson : POINTER TO JsonType; 
	_i: INT;
	pString: POINTER TO BYTE;
END_VAR
IF NOT _bInit AND NOT _barr AND NOT _AddKey THEN 
	RETURN; 
END_IF
pJson := CreateJsonType(); 
pJson^.DataType := JSONDATATYPE.JSON_DATA_STRING; 
_i := 0;
WHILE value[_i] <> 0 DO
	_i := _i + 1; 
END_WHILE
pString := __NEW(BYTE,_i); 
_i := 0; 
WHILE value[_i] <> 0 DO 
	pString[_i] := value[_i]; 
	_i := _i + 1; 
END_WHILE
pString[_i] := 0; 
pJson^.pValue := pString; 
IF NOT _bArr THEN 
	_arrObjects[_objIdx]^.Put(_key,pJson); 
	_AddKey := FALSE; 
ELSE 
	_arrArrays[_arrIdx]^.PushBack(ADR(pJson)); 
END_IF
END_METHOD

METHOD AddUdint
VAR_INPUT
  value : UDINT;
END_VAR
VAR
	
	pJson: Pointer TO JsonType;
	pDint: POINTER TO UDINT;
END_VAR
IF NOT _bInit AND NOT _barr AND NOT _AddKey THEN 
	RETURN; 
END_IF
pJson := CreateJsonType(); 
pJson^.DataType := JSONDATATYPE.JSON_DATA_INT; 
pDint := __NEW(UDINT); 
pDint^ := value;
pJson^.pValue := pDint; 
IF NOT _bArr THEN 
	_arrObjects[_objIdx]^.Put(_key,pJson); 
	_AddKey := FALSE; 
ELSE 
	_arrArrays[_arrIdx]^.PushBack(ADR(pJson)); 
END_IF
END_METHOD

METHOD PRIVATE Clean : BOOL
VAR_INPUT
END_VAR
VAR 
	arrIdx : INT;  
	pJsonData: POINTER TO JsonTYPE;
	pJsonManager: Pointer TO JsonObjectManager;
	pString: POINTER TO BYTE;
	pBackingLists : Pointer TO DynamicJsonTypeContainer;
END_VAR
arrIdx := 0; 
WHILE _lCreatedValues.GetIterator().Next(ADR(pJsonData)) DO 
	IF pJsonData <> 0 THEN 
		DeleteJsonNode(pJsonData); 
	END_IF
	pJsonData := 0; 
END_WHILE
WHILE _lCreatedKeys.GetIterator().Next(ADR(pString)) DO 
	IF pString <> 0 THEN
		__DELETE(pString);
	END_IF 
	pString := 0;  
END_WHILE
WHILE _lCreatedObj.GetIterator().Next(ADR(pJsonManager)) DO
	pJsonManager^.Destroy(); 
	__DELETE(pJsonManager); 
END_WHILE
WHILE lCreatedLists.GetIterator().Next(ADR(pBackingLists)) DO 
	__DELETE(pBackingLists); 
END_WHILE
_lCreatedValues.Clear(); 
_lCreatedObj.Clear(); 
_lCreatedKeys.Clear(); 
lCreatedLists.Clear();
END_METHOD

METHOD CopyDocument : UDINT
VAR_IN_OUT CONSTANT
  pDoc       : STRING;
END_VAR
VAR_INPUT
  nDoc       : UDINT;
  bPretty : BOOL := FALSE; 
END_VAR
VAR_OUTPUT
  hrErrorCode:PVOID;
END_VAR
VAR
	_bytePtr : POINTER TO BYTE; 
	_i: UDINT;
	_Settings : JsonSerializeConfig;
END_VAR
IF NOT _bInit THEN 
	Init(); 
END_IF
_bytePtr := ADR(pDoc); 
_settings.PrettyPrint := bPretty;
_settings.IndentSize := 4; 
CopyDocument := TO_UDINT(JsonSerializer(GetRoot(),ADR(pDoc),TO_DINT(nDoc),_settings));
END_METHOD

METHOD PRIVATE CreateArray : POINTER TO DynamicList
VAR_INPUT
END_VAR

VAR
	_pBacking: POINTER TO DynamicJsonTypeContainer;
	_lArray: POINTER TO DynamicList;
END_VAR
_pBacking := __NEW(DynamicJsonTypeContainer(udSize := 1)); 
lCreatedLists.PushBack(ADR(_pBacking)); 
_lArray := __NEW(DynamicList); 
_lArray^(DataContainer := _pBacking^); 
CreateArray := _lArray;
END_METHOD

METHOD PRIVATE CreateJsonType : POINTER TO JSONType
VAR_INPUT
END_VAR

VAR
	_pJsonType: POINTER TO JsonType;
END_VAR
_pJsonType := __NEW(JsonType); 
_lCreatedValues.PushBack(ADR(_pJsonType)); 
CreateJsonType := _pJsonType;
END_METHOD

METHOD PRIVATE CreateObj : Pointer TO JsonObjectManager
VAR_INPUT
END_VAR

VAR
	pJsonManager: POINTER TO JsonObjectManager;
END_VAR
pJsonManager := __NEW(JsonObjectManager); 
pJsonManager^.Create(); 
_lCreatedObj.PushBack(ADR(pJsonManager));
CreateObj := pJsonManager; 
_bInit := TRUE;
END_METHOD

METHOD PRIVATE DeleteJsonNode : BOOL
VAR_INPUT
	pJsonNode : POINTER TO JSONTYPE; 
END_VAR
VAR
	pString : POINTER TO STRING; 
	pLINT  : POINTER TO DINT; 
	pBOOL  : POINTER TO BOOL; 
	pFloat : POINTER TO REAL; 
	pJasonType : POINTER TO JsonType; 
	pJsonArray : POINTER TO DynamicList; 
END_VAR
IF pJsonNode = 0 THEN 
	RETURN; 
END_IF
CASE pJsonNode^.DataType OF 
	JSON_DATA_NULL: 
// nothing to clean	
    JSON_DATA_BOOL: 
		pBool := pJsonNode^.pValue; 
		__DELETE(pBool);
    JSON_DATA_INT:
		pLINT := pJsonNode^.pValue;
		__DELETE(pLINT); 
    JSON_DATA_REAL: 
		pFloat := pJsonNode^.pValue; 
		__DELETE(pFloat);
    JSON_DATA_STRING: 
		pString :=pJsonNode^.pValue;
		__DELETE(pString); 
	JSON_DATA_ARRAY:
		pJsonArray := pJsonNode^.pValue; 
		__DELETE(pJsonArray); 
END_CASE
	__DELETE(pJsonNode);
END_METHOD

METHOD EndArray 
VAR_INPUT
END_VAR
IF NOT _bInit THEN
	Init(); 
END_IF
_arrIdx := _arrIdx - 1; 
IF _arrIdx < 0 THEN
	_bArr := FALSE; 
	_AddKey := FALSE; 
END_IF
END_METHOD

METHOD EndObject 
VAR_INPUT
END_VAR

VAR

END_VAR
IF NOT _bInit THEN
	Init(); 
END_IF
_AddKey := FALSE; 
_ObjIdx := _ObjIdx - 1;
END_METHOD

METHOD GetRoot : POINTER TO JsonType
VAR_INPUT
END_VAR
VAR
	pJson : POINTER TO JsonObjectManager; 
END_VAR
IF NOT _bInit THEN
	Init(); 
END_IF
pJson := _root.pValue; 
GetRoot := pJson^.GetValue('root');
END_METHOD

METHOD PRIVATE Init : BOOL
VAR_INPUT
END_VAR
_root.DataType := JSONDATATYPE.JSON_DATA_OBJECT; 
_root.pValue := CreateObj(); 
_arrObjects[0] := _root.pValue;  
_bInit := TRUE; 
_arrIdx := -1; 
_objIdx := 0;
_bRootAdded := FALSE;
END_METHOD

METHOD ResetDocument 
VAR_INPUT
END_VAR
Clean(); 
_bInit :=FALSE; 
_AddKey:=FALSE;
_bRootAdded :=FALSE; 
_arrIdx := -1; 
_objIdx := 0;
END_METHOD

METHOD StartArray  
VAR_INPUT
END_VAR
VAR
	pJson : POINTER TO JSONTYPE; 
	pArr: POINTER TO DynamicList;
END_VAR
IF NOT _bInit THEN
	Init(); 
END_IF
IF NOT _bRootAdded THEN 
	AddKey('root'); 
	_bRootAdded := TRUE; 
END_IF
IF NOT _barr AND NOT _AddKey THEN 
	RETURN; 
END_IF
_arrIdx := _arrIdx + 1; 
pJson := CreateJsonType(); 
pJson^.DataType := JSONDATATYPE.JSON_DATA_ARRAY; 
pArr := CreateArray();
pJson^.pValue := pArr; 
IF NOT _bArr THEN 
	_arrObjects[_objIdx]^.Put(_key,pJson); 
	_AddKey := FALSE; 
ELSE 
	_arrArrays[_arrIdx-1]^.PushBack(ADR(pJson)); 
END_IF
_arrArrays[_arrIdx] := pArr; 
_bArr := TRUE;
END_METHOD

METHOD StartObject 
VAR_INPUT
END_VAR

VAR

	pJson: POINTER TO JsonType;
	pObj: POINTER TO JsonObjectManager;
END_VAR
IF NOT _bInit THEN
	Init(); 
END_IF
IF NOT _bRootAdded THEN 
	AddKey('root'); 
	_bRootAdded := TRUE; 
END_IF
IF NOT _barr AND NOT _AddKey THEN 
	RETURN; 
END_IF 
pJson := CreateJsonType(); 
pJson^.DataType := JSONDATATYPE.JSON_DATA_Object; 
pObj := CreateObj();
pJson^.pValue := pObj; 
IF NOT _bArr THEN 
	_arrObjects[_objIdx]^.Put(_key,pJson); 
	_AddKey := FALSE; 
ELSE 
	_arrArrays[_arrIdx]^.PushBack(ADR(pJson)); 
END_IF
_objIdx := _objIdx + 1; 
_arrObjects[_objIdx] := pObj;
END_METHOD

END_FUNCTION_BLOCK

// Device/Application/GetJsonNodeByKey
FUNCTION GetJsonNodeByKey: Pointer TO JsonType; 
VAR_INPUT
	strKey : STRING; 
END_VAR
VAR_IN_OUT
	pDoc : POINTER TO JsonObject; 
END_VAR
VAR_OUTPUT
END_VAR
VAR
	i: INT;
	pStr : POINTER TO STRING; 
END_VAR

	GetJsonNodeByKey := 0; 
IF pDoc = 0 THEN 
	RETURN; 
END_IF
IF pDoc^.iNumValues <1 THEN
	RETURN; 
END_IF
FOR i := 0 TO pDoc^.iNumValues - 1 DO 
	pStr := pDoc^.pKeys[i]^.pValue; 
	IF pStr^ = strKey THEN 
		GetJsonNodeByKey := pDoc^.pValues[i];
		RETURN;  
	END_IF
END_FOR

END_FUNCTION

// Device/Application/GetNodeAsObject
FUNCTION GetNodeAsObject : POINTER TO JsonObject
VAR_INPUT
	pJsonNode : POINTER TO JsonType;
END_VAR
VAR_OUTPUT

END_VAR
VAR
END_VAR

GetNodeAsObject := 0; 
IF pJsonNode = 0 THEN 
	RETURN; 
END_IF
IF pJsonNode^.DataType <> JsonDataType.JSON_DATA_OBJECT THEN 
	RETURN; 
END_IF
GetNodeAsObject := pJsonNode^.pValue;

END_FUNCTION

// Device/Application/isJsonNodeNull
FUNCTION isJsonNodeNull : BOOL
VAR_INPUT
	pJsonNode : POINTER TO JsonType; 
END_VAR
VAR
END_VAR

isJsonNodeNull := TRUE; 
IF pJsonNode = 0 THEN
	RETURN;
END_IF
IF pJsonNode^.DataType = JSONDataType.JSON_DATA_NULL THEN 
	RETURN; 
END_IF
isJsonNodeNull := FALSE;

END_FUNCTION

// Device/Application/JsonDomParser
FUNCTION_BLOCK JsonDomParser
VAR
 _parser : JsonParser2; 
 _doc : POINTER TO JsonObject; 
 _node : POINTER TO JsonType; 
END_VAR

METHOD CopyJson :UDINT
VAR_INPUT
  v    : POINTER TO JsonType;
  pDoc : POINTER to BYTE;
  nDoc : UDINT;
END_VAR
VAR
	Settings : JsonSerializeConfig;
END_VAR
CopyJson := TO_UDINT(JsonSerializer(v, pDoc,TO_DINT(nDoc),Settings));
END_METHOD

METHOD CopyString : UDINT
VAR_INPUT
  v    : POINTER TO JsonType;
  pStr : POINTER TO BYTE;
  nStr : UDINT;
END_VAR
VAR
	size: UDINT;
END_VAR
GetNodeAsString(v,pstr,nStr,retStrSize => size); 
CopyString := size;
END_METHOD

//FB_Exit must be implemented explicitly. If there is an implementation, then the
//method is called before the controller removes the code of the function block instance
//(implicit call). The return value is not evaluated.
METHOD FB_Exit: BOOL
VAR_INPUT
    bInCopyCode: BOOL;  // TRUE: the exit method is called in order to leave the instance which will be copied afterwards (online change).  
END_VAR
_parser.Clean();
END_METHOD

METHOD FindMember : POINTER TO JsonType; 
VAR_INPUT
  v      : POINTER TO JsonType;
END_VAR
VAR_IN_OUT CONSTANT
  member : STRING;
END_VAR
VAR
END_VAR
FindMember := GetJsonNodeByKey(Member,v);
END_METHOD

METHOD GetArrayValueByIdx : POINTER TO JsonType
VAR_INPUT
  v   : POINTER TO JsonType;
  idx : UDINT;
END_VAR
GetArrayValueByIdx := GetNodeAtIndex(v,idx);
END_METHOD

METHOD GetBool : BOOL
VAR_INPUT
  v : POINTER TO JSONType;
END_VAR
VAR
	bValue :BOOL; 
	bSuccess: BOOL;
END_VAR
bSuccess := GetNodeAsBool(v,bJsonVal => bValue); 
GetBool := bValue and bSuccess;
END_METHOD

METHOD GetInt : DINT
VAR_INPUT
  v : POINTER TO JsonType;
END_VAR
VAR
	t_Dint: DINT;
	bSuccess: BOOL;
END_VAR
bSuccess := GetNodeAsInt(v,iJsonVal => t_Dint); 
IF bSuccess THEN 
	GetInt := t_Dint; 
END_IF
END_METHOD

METHOD GetReal : Real
VAR_INPUT
	  v : POINTER TO JSONType;
END_VAR

VAR
	rValue: REAL;
END_VAR
GetNodeAsReal(v,rJsonVal => rValue); 
GetReal := rValue;
END_METHOD

METHOD GetString : STRING(255)
VAR_INPUT
  v : POINTER TO JsonType;
END_VAR
VAR
	bytes : ARRAY[0..256] OF BYTE; 
	pString : POINTER TO STRING(255); 
END_VAR
pString := ADR(bytes); 
GetNodeAsString(v,pString,256); 
GetString := pString^;
END_METHOD

METHOD isNull : BOOL
VAR_INPUT
	v : POINTER TO JSONType;
END_VAR
isNull := isJsonNodeNull(v);
END_METHOD

METHOD ParseDocument : POINTER TO JsonType
VAR_INPUT
	udSize : UDINT;
END_VAR
VAR_IN_OUT CONSTANT
  sJson : STRING;
END_VAR
ParseDocument := 0; 
IF(_parser.Parse(ADR(sJson),udSize)) THEN 
	ParseDocument := _parser.GetRootDoc(); 
END_IF
END_METHOD

METHOD ResetDocument : BOOL
VAR_INPUT
END_VAR
_parser.Clean();
END_METHOD

END_FUNCTION_BLOCK

// Device/Application/JsonParser
FUNCTION_BLOCK JsonParser
VAR_INPUT
	MAX_DOC_DEPTH : INT; 
	MAX_DOC_WIDTH : INT; 
END_VAR
VAR_OUTPUT
END_VAR
VAR
	root : JsonType;
END_VAR

METHOD Clean : BOOL
VAR_INPUT
	
END_VAR
VAR
	arrObjects : ARRAY[0..Parameters.MAX_DOC_DEPTH] OF POINTER TO JsonObject; 
	arrArrays  : ARRAY[0..Parameters.MAX_DOC_DEPTH] OF POINTER TO JsonArray; 
	objIdx : INT; 
	arrIdx : INT;  
	curObjIdx : ARRAY[0.. Parameters.MAX_DOC_DEPTH] OF INT; 
	j: LINT;
	i: LINT; 
END_VAR
arrObjects[0] := root.pValue;
IF arrObjects[0] = 0 THEN 
	RETURN;
END_IF 
IF arrObjects[0]^.iNumValues = 0 THEN 
	Return; 
END_IF
objIdx := 0; 
arrIdx := 0; 
WHILE TRUE DO
	IF curObjIdx[objIdx] = arrObjects[ObjIdx]^.iNumValues THEN 	
		__DELETE(arrObjects[ObjIdx]^.pKeys); 
		__DELETE(arrObjects[ObjIdx]^.pValues); 
		__DELETE(arrObjects[objIdx]); 
		objIdx := objIdx - 1;
		IF objIdx < 0 THEN 
			EXIT; 
		END_IF 
		CONTINUE; 
	END_IF
	CASE arrObjects[objIdx]^.pValues[curObjIdx[objIdx]]^.DataType OF 
    JSON_DATA_ARRAY:
 		arrArrays[arrIdx] := arrObjects[objIdx]^.pValues[curObjIdx[objIdx]]^.pValue;
		arrIdx := arrIdx+ 1; 
		THIS^.DeleteJsonNode(arrObjects[objIdx]^.pValues[curObjIdx[objIdx]]); 
		THIS^.DeleteJsonNode(arrObjects[objIdx]^.pKeys[curObjIdx[objIdx]]); 
		curObjIdx[objIdx] := curObjIdx[objIdx] + 1; 
    JSON_DATA_OBJECT: 
		arrObjects[objIdx + 1] :=  arrObjects[objIdx]^.pValues[curObjIdx[objIdx]]^.pValue; 
		THIS^.DeleteJsonNode(arrObjects[objIdx]^.pValues[curObjIdx[objIdx]]); 
		THIS^.DeleteJsonNode(arrObjects[objIdx]^.pKeys[curObjIdx[objIdx]]); 
		curObjIdx[objIdx] := curObjIdx[objIdx] + 1;  
		objIdx := objIdx + 1; 
	ELSE
		THIS^.DeleteJsonNode(arrObjects[objIdx]^.pValues[curObjIdx[objIdx]]); 
		THIS^.DeleteJsonNode(arrObjects[objIdx]^.pKeys[curObjIdx[objIdx]]); 
		curObjIdx[objIdx] := curObjIdx[objIdx] + 1; 
	END_CASE
END_WHILE
IF arrIdx = 0 THEN 
	RETURN; 
END_IF
FOR i := 0 TO arrIdx - 1 DO 
	IF arrArrays[i]^.iNumValues = 0 THEN 
		RETURN; 
	END_IF
	FOR j:= 0 TO arrArrays[i]^.iNumValues -1 DO 
		THIS^.DeleteJsonNode(arrArrays[i]^.Values[j]); 
	END_FOR
	__DELETE(arrArrays[i]^.Values); 
	__DELETE(arrArrays[i]); 
END_FOR
END_METHOD

METHOD PRIVATE DeleteJsonNode : BOOL
VAR_INPUT
	pJsonNode : POINTER TO JSONTYPE; 
END_VAR
VAR
	pString : POINTER TO STRING; 
	pLINT  : POINTER TO DINT; 
	pBOOL  : POINTER TO BOOL; 
	pFloat : POINTER TO REAL; 
	pJasonType : POINTER TO JsonType; 
END_VAR
IF pJsonNode = 0 THEN 
	RETURN; 
END_IF
CASE pJsonNode^.DataType OF 
	JSON_DATA_NULL: 
// nothing to clean	
    JSON_DATA_BOOL: 
		pBool := pJsonNode^.pValue; 
		__DELETE(pBool);
    JSON_DATA_INT:
		pLINT := pJsonNode^.pValue;
		__DELETE(pLINT); 
    JSON_DATA_REAL: 
		pFloat := pJsonNode^.pValue; 
		__DELETE(pFloat);
    JSON_DATA_STRING: 
		pString :=pJsonNode^.pValue;
		__DELETE(pString); 
	
END_CASE
	__DELETE(pJsonNode);
END_METHOD

//FB_Exit must be implemented explicitly. If there is an implementation, then the
//method is called before the controller removes the code of the function block instance
//(implicit call). The return value is not evaluated.
METHOD  FB_Exit: BOOL
VAR_INPUT
    bInCopyCode: BOOL;  // TRUE: the exit method is called in order to leave the instance which will be copied afterwards (online change).  
END_VAR
This^.Clean();
END_METHOD

METHOD GetRootDoc : POINTER TO JsonObject; 
VAR_INPUT
END_VAR
VAR
	pJson : POINTER TO JsonObject; 
	pJsonType : POINTER TO JsonType; 
END_VAR
pJson := root.pValue; 
IF pJSON = 0 THEN 
	RETURN; 
END_IF
IF pJson^.iNumValues = 1 AND pJson^.pKeys[0] = 0 AND pJson^.pValues <> 0 THEN 
	pJsonType := pJson^.pValues[0]; 
	GetRootDoc := pJsonType^.pValue; 
ELSE 
	GetRootDoc := pJson; 
END_IF
END_METHOD

METHOD Parse : BOOL
VAR_INPUT
	pJsonStr : POINTER TO BYTE; 
	StrSize  : LINT; 
END_VAR
VAR
	Offset : LINT; 
	stJsonToken: JsonToken;
	arrObjects : ARRAY[0..Parameters.MAX_DOC_DEPTH] OF POINTER TO JsonObject; 
	arrArrays  : ARRAY[0..Parameters.MAX_DOC_DEPTH] OF POINTER TO JsonArray; 
	objIdx : INT; 
	arrIdx : INT; 
	curArrIdx : ARRAY[0.. Parameters.MAX_DOC_DEPTH] OF INT; 
	curObjIdx : ARRAY[0.. Parameters.MAX_DOC_DEPTH] OF INT; 
	arrStartObjIdx : INT; 
	bArr : BOOL; 
	bArObj : BOOL; 
	pBool: POINTER TO BOOL;
	bNeedKey : BOOL; 
	HasDecimal: BOOL;
	jsonNodeVal: JsonType;
	pJsonObj: POINTER TO JSONObject;
	iArrDepth : INT; 
	pJsonArray: POINTER TO JSONARRAY;
	pJsonType: POINTER TO JSONType;
	bFirstObj: BOOL;
	pRootOBJ: POINTER TO JSONObject;
END_VAR
THIS^.Clean(); 
Offset := 0; 
objIdx := 0; 
arrIdx := -1; 
THIS^.root.DataType := JsonDataType.JSON_DATA_OBJECT;
pRootOBJ := __NEW(JSONObject); 
THIS^.root.pValue := pRootObj; 
arrObjects[0] := pRootObj; 
pRootObj^.pKeys := __NEW(POINTER TO JSONType, PARAMETERS.MAX_ARR_SIZE); 
pRootObj^.pValues := __NEW(POINTER TO JSONTYpe, PARAMETERS.MAX_ARR_SIZE); 
bArr := FALSE; 
bNeedKey := TRUE; 
bFirstObj := TRUE; 
WHILE Offset < StrSize DO 
	stJsonToken := GetNextJsonToken(pJsonStr,StrSize, Offset := Offset); 
	CASE stJsonToken.TokenType OF 
		JSON_TOKEN_NULL, JSON_TOKEN_TRUE, JSON_TOKEN_FALSE, JSON_TOKEN_NUMBER:
			jsonNodeVal := JsonHadlr(pJsonStr,stJsonToken);
			IF bARR AND NOT bARObj THEN 
				arrArrays[arrIdx]^.Values[curArrIdx[arridx]] := __NEW(JSONType); 
				arrArrays[arrIdx]^.Values[curArrIdx[arridx]]^ := jsonNodeVal; 
				curArrIdx[arridx] := curArrIdx[arridx] + 1; 
			ELSE 
				arrObjects[objIdx]^.pValues[curObjIdx[objIdx]]:=  __NEW(JSONType);
				arrObjects[objIdx]^.pValues[curObjIdx[objIdx]]^:= jsonNodeVal; 
				curObjIdx[objIdx] := curObjIdx[objIdx] + 1;
				bNeedKey := TRUE;  
			END_IF
		JSON_TOKEN_STRING: 
			jsonNodeVal := JsonHadlr(pJsonStr,stJsonToken);
			IF bNeedKey THEN 
				arrObjects[objIdx]^.pKeys[curObjIdx[objIdx]] := __NEW(JSONType); 
				arrObjects[objIdx]^.pKeys[curObjIdx[objIdx]]^ := jsonNodeVal; 
				bNeedKey := FALSE; 
			ELSIF bArr THEN 
				arrArrays[arrIdx]^.Values[curArrIdx[arridx]] := __NEW(JSONType); 
				arrArrays[arrIdx]^.Values[curArrIdx[arridx]]^ := jsonNodeVal; 
				curArrIdx[arridx] := curArrIdx[arridx]+1;
			ELSE
				arrObjects[objIdx]^.pValues[curObjIdx[objIdx]] := __NEW(JSONType); 
				arrObjects[objIdx]^.pValues[curObjIdx[objIdx]]^ := jsonNodeVal;
				curObjIdx[objIdx] := curObjIdx[objIdx] + 1; 
				bNeedKey := TRUE; 
			END_IF
    	JSON_TOKEN_LBRACE:      // {
			pJsonObj := __NEW(JSONObject); 
			pJsonObj^.pKeys := __NEW(POINTER TO JsonType, PARAMETERS.MAX_ARR_SIZE);
			pJsonObj^.pValues := __NEW(POINTER TO JsonType, PARAMETERS.MAX_ARR_SIZE);  
			pJsonType := __NEW(JSONType); 
			pJsonType^.pValue := pJsonObj; 
			pJsonType^.DataType :=JsonDataType.JSON_DATA_OBJECT;  
			IF bARR THEN 
				arrArrays[arrIdx]^.Values[curArrIdx[arridx]] := pJsonType; 
				bArObj := TRUE; 
				curArrIdx[arridx] := curArrIdx[arridx] + 1; 
			ELSE
				arrObjects[objIdx]^.pValues[curObjIdx[objIdx]] := pJsonType; 
				curObjIdx[objIdx] := curObjIdx[objIdx] + 1; 
			END_IF
			
			objIdx := objIdx + 1; 
			arrObjects[objIdx] := pJsonObj;
			bNeedKey := TRUE;  
			
    	JSON_TOKEN_RBRACE:      // }
			arrObjects[objIdx]^.iNumValues := curObjIdx[objIdx]; 
			curObjIdx[objIdx] := 0; 
			objIdx := objIdx - 1; 
			bArObj := FALSE; 
			
    	JSON_TOKEN_LBRACKET:    // [
			pJsonArray := __NEW(JSONARRAY);
			pJsonArray^.Values := __NEW(POINTER TO JsonType,PARAMETERS.MAX_ARR_SIZE);  
			arrIdx := arrIdx + 1; 
			arrArrays[arrIdx] := pJsonArray; 
			IF bArr THEN 
				iArrDepth := iArrDepth + 1; 
				arrArrays[arrIdx -iarrDepth]^.Values[curArrIdx[arridx-iarrDepth]] := pJsonArray; 
			ELSE
				arrObjects[objIdx]^.pValues[curObjIdx[objIdx]] := __NEW(JsonType); 
				arrObjects[objIdx]^.pValues[curObjIdx[objidx]]^.pValue := pJsonArray; 
				arrObjects[objIdx]^.pValues[curObjIdx[objidx]]^.DataType := JsonDataType.JSON_DATA_ARRAY; 
				curObjIdx[objIdx] :=  curObjIdx[objIdx] + 1;
			END_IF
			bArr := TRUE; 
			bNeedKey := FALSE; 
			
    	JSON_TOKEN_RBRACKET:    // ]
			arrArrays[arrIdx]^.iNumValues := curArrIdx[arridx]; 
			curArrIdx[arridx] := 0; 
			arrIdx := arrIdx - 1; 
			iArrDepth := iArrDepth - 1; 
			IF iArrDepth < 0 THEN 
				iArrDepth := 0; 
				bArr := FALSE;
				bNeedKey := TRUE; 
			END_IF
			 
			
    	JSON_TOKEN_COMMA:       // ,
		
    	JSON_TOKEN_COLON:       // :
		
    	JSON_TOKEN_EOF:
			arrObjects[0]^.iNumValues := curObjIdx[0]; 
			EXIT; 
    	JSON_TOKEN_ERROR: 
			EXIT; 
	END_CASE
END_WHILE
END_METHOD

END_FUNCTION_BLOCK

